   // UNICODE_TO_GBK[34826] := 16#8F38;
   // UNICODE_TO_GBK[34827] := 16#DD94;
   // UNICODE_TO_GBK[34828] := 16#8F39;
   // UNICODE_TO_GBK[34829] := 16#DD95;
   // UNICODE_TO_GBK[34830] := 16#8F3A;
   // UNICODE_TO_GBK[34831] := 16#DD96;
   // UNICODE_TO_GBK[34832] := 16#8F3B;
   // UNICODE_TO_GBK[34833] := 16#DD97;
   // UNICODE_TO_GBK[34834] := 16#8F3C;
   // UNICODE_TO_GBK[34835] := 16#DD98;
   // UNICODE_TO_GBK[34836] := 16#8F3D;
   // UNICODE_TO_GBK[34837] := 16#DD99;
   // UNICODE_TO_GBK[34838] := 16#8F3E;
   // UNICODE_TO_GBK[34839] := 16#DD9A;
   // UNICODE_TO_GBK[34840] := 16#8F3F;
   // UNICODE_TO_GBK[34841] := 16#DD9B;
   // UNICODE_TO_GBK[34842] := 16#8F40;
   // UNICODE_TO_GBK[34843] := 16#DD9C;
   // UNICODE_TO_GBK[34844] := 16#8F41;
   // UNICODE_TO_GBK[34845] := 16#DD9D;
   // UNICODE_TO_GBK[34846] := 16#8F42;
   // UNICODE_TO_GBK[34847] := 16#DD9E;
   // UNICODE_TO_GBK[34848] := 16#8F43;
   // UNICODE_TO_GBK[34849] := 16#DD9F;
   // UNICODE_TO_GBK[34850] := 16#8F44;
   // UNICODE_TO_GBK[34851] := 16#DDA0;
   // UNICODE_TO_GBK[34852] := 16#8F45;
   // UNICODE_TO_GBK[34853] := 16#DE40;
   // UNICODE_TO_GBK[34854] := 16#8F46;
   // UNICODE_TO_GBK[34855] := 16#DE41;
   // UNICODE_TO_GBK[34856] := 16#8F47;
   // UNICODE_TO_GBK[34857] := 16#DE42;
   // UNICODE_TO_GBK[34858] := 16#8F48;
   // UNICODE_TO_GBK[34859] := 16#DE43;
   // UNICODE_TO_GBK[34860] := 16#8F49;
   // UNICODE_TO_GBK[34861] := 16#DE44;
   // UNICODE_TO_GBK[34862] := 16#8F4A;
   // UNICODE_TO_GBK[34863] := 16#DE45;
   // UNICODE_TO_GBK[34864] := 16#8F4B;
   // UNICODE_TO_GBK[34865] := 16#DE46;
   // UNICODE_TO_GBK[34866] := 16#8F4C;
   // UNICODE_TO_GBK[34867] := 16#DE47;
   // UNICODE_TO_GBK[34868] := 16#8F4D;
   // UNICODE_TO_GBK[34869] := 16#DE48;
   // UNICODE_TO_GBK[34870] := 16#8F4E;
   // UNICODE_TO_GBK[34871] := 16#DE49;
   // UNICODE_TO_GBK[34872] := 16#8F4F;
   // UNICODE_TO_GBK[34873] := 16#DE4A;
   // UNICODE_TO_GBK[34874] := 16#8F50;
   // UNICODE_TO_GBK[34875] := 16#DE4B;
   // UNICODE_TO_GBK[34876] := 16#8F51;
   // UNICODE_TO_GBK[34877] := 16#DE4C;
   // UNICODE_TO_GBK[34878] := 16#8F52;
   // UNICODE_TO_GBK[34879] := 16#DE4D;
   // UNICODE_TO_GBK[34880] := 16#8F53;
   // UNICODE_TO_GBK[34881] := 16#DE4E;
   // UNICODE_TO_GBK[34882] := 16#8F54;
   // UNICODE_TO_GBK[34883] := 16#DE4F;
   // UNICODE_TO_GBK[34884] := 16#8F55;
   // UNICODE_TO_GBK[34885] := 16#DE50;
   // UNICODE_TO_GBK[34886] := 16#8F56;
   // UNICODE_TO_GBK[34887] := 16#DE51;
   // UNICODE_TO_GBK[34888] := 16#8F57;
   // UNICODE_TO_GBK[34889] := 16#DE52;
   // UNICODE_TO_GBK[34890] := 16#8F58;
   // UNICODE_TO_GBK[34891] := 16#DE53;
   // UNICODE_TO_GBK[34892] := 16#8F59;
   // UNICODE_TO_GBK[34893] := 16#DE54;
   // UNICODE_TO_GBK[34894] := 16#8F5A;
   // UNICODE_TO_GBK[34895] := 16#DE55;
   // UNICODE_TO_GBK[34896] := 16#8F5B;
   // UNICODE_TO_GBK[34897] := 16#DE56;
   // UNICODE_TO_GBK[34898] := 16#8F5C;
   // UNICODE_TO_GBK[34899] := 16#DE57;
   // UNICODE_TO_GBK[34900] := 16#8F5D;
   // UNICODE_TO_GBK[34901] := 16#DE58;
   // UNICODE_TO_GBK[34902] := 16#8F5E;
   // UNICODE_TO_GBK[34903] := 16#DE59;
   // UNICODE_TO_GBK[34904] := 16#8F5F;
   // UNICODE_TO_GBK[34905] := 16#DE5A;
   // UNICODE_TO_GBK[34906] := 16#8F60;
   // UNICODE_TO_GBK[34907] := 16#DE5B;
   // UNICODE_TO_GBK[34908] := 16#8F61;
   // UNICODE_TO_GBK[34909] := 16#DE5C;
   // UNICODE_TO_GBK[34910] := 16#8F62;
   // UNICODE_TO_GBK[34911] := 16#DE5D;
   // UNICODE_TO_GBK[34912] := 16#8F63;
   // UNICODE_TO_GBK[34913] := 16#DE5E;
   // UNICODE_TO_GBK[34914] := 16#8F64;
   // UNICODE_TO_GBK[34915] := 16#DE5F;
   // UNICODE_TO_GBK[34916] := 16#8F65;
   // UNICODE_TO_GBK[34917] := 16#DE60;
   // UNICODE_TO_GBK[34918] := 16#8F66;
   // UNICODE_TO_GBK[34919] := 16#B3B5;
   // UNICODE_TO_GBK[34920] := 16#8F67;
   // UNICODE_TO_GBK[34921] := 16#D4FE;
   // UNICODE_TO_GBK[34922] := 16#8F68;
   // UNICODE_TO_GBK[34923] := 16#B9EC;
   // UNICODE_TO_GBK[34924] := 16#8F69;
   // UNICODE_TO_GBK[34925] := 16#D0F9;
   // UNICODE_TO_GBK[34926] := 16#8F6A;
   // UNICODE_TO_GBK[34927] := 16#DE61;
   // UNICODE_TO_GBK[34928] := 16#8F6B;
   // UNICODE_TO_GBK[34929] := 16#E9ED;
   // UNICODE_TO_GBK[34930] := 16#8F6C;
   // UNICODE_TO_GBK[34931] := 16#D7AA;
   // UNICODE_TO_GBK[34932] := 16#8F6D;
   // UNICODE_TO_GBK[34933] := 16#E9EE;
   // UNICODE_TO_GBK[34934] := 16#8F6E;
   // UNICODE_TO_GBK[34935] := 16#C2D6;
   // UNICODE_TO_GBK[34936] := 16#8F6F;
   // UNICODE_TO_GBK[34937] := 16#C8ED;
   // UNICODE_TO_GBK[34938] := 16#8F70;
   // UNICODE_TO_GBK[34939] := 16#BAE4;
   // UNICODE_TO_GBK[34940] := 16#8F71;
   // UNICODE_TO_GBK[34941] := 16#E9EF;
   // UNICODE_TO_GBK[34942] := 16#8F72;
   // UNICODE_TO_GBK[34943] := 16#E9F0;
   // UNICODE_TO_GBK[34944] := 16#8F73;
   // UNICODE_TO_GBK[34945] := 16#E9F1;
   // UNICODE_TO_GBK[34946] := 16#8F74;
   // UNICODE_TO_GBK[34947] := 16#D6E1;
   // UNICODE_TO_GBK[34948] := 16#8F75;
   // UNICODE_TO_GBK[34949] := 16#E9F2;
   // UNICODE_TO_GBK[34950] := 16#8F76;
   // UNICODE_TO_GBK[34951] := 16#E9F3;
   // UNICODE_TO_GBK[34952] := 16#8F77;
   // UNICODE_TO_GBK[34953] := 16#E9F5;
   // UNICODE_TO_GBK[34954] := 16#8F78;
   // UNICODE_TO_GBK[34955] := 16#E9F4;
   // UNICODE_TO_GBK[34956] := 16#8F79;
   // UNICODE_TO_GBK[34957] := 16#E9F6;
   // UNICODE_TO_GBK[34958] := 16#8F7A;
   // UNICODE_TO_GBK[34959] := 16#E9F7;
   // UNICODE_TO_GBK[34960] := 16#8F7B;
   // UNICODE_TO_GBK[34961] := 16#C7E1;
   // UNICODE_TO_GBK[34962] := 16#8F7C;
   // UNICODE_TO_GBK[34963] := 16#E9F8;
   // UNICODE_TO_GBK[34964] := 16#8F7D;
   // UNICODE_TO_GBK[34965] := 16#D4D8;
   // UNICODE_TO_GBK[34966] := 16#8F7E;
   // UNICODE_TO_GBK[34967] := 16#E9F9;
   // UNICODE_TO_GBK[34968] := 16#8F7F;
   // UNICODE_TO_GBK[34969] := 16#BDCE;
   // UNICODE_TO_GBK[34970] := 16#8F80;
   // UNICODE_TO_GBK[34971] := 16#DE62;
   // UNICODE_TO_GBK[34972] := 16#8F81;
   // UNICODE_TO_GBK[34973] := 16#E9FA;
   // UNICODE_TO_GBK[34974] := 16#8F82;
   // UNICODE_TO_GBK[34975] := 16#E9FB;
   // UNICODE_TO_GBK[34976] := 16#8F83;
   // UNICODE_TO_GBK[34977] := 16#BDCF;
   // UNICODE_TO_GBK[34978] := 16#8F84;
   // UNICODE_TO_GBK[34979] := 16#E9FC;
   // UNICODE_TO_GBK[34980] := 16#8F85;
   // UNICODE_TO_GBK[34981] := 16#B8A8;
   // UNICODE_TO_GBK[34982] := 16#8F86;
   // UNICODE_TO_GBK[34983] := 16#C1BE;
   // UNICODE_TO_GBK[34984] := 16#8F87;
   // UNICODE_TO_GBK[34985] := 16#E9FD;
   // UNICODE_TO_GBK[34986] := 16#8F88;
   // UNICODE_TO_GBK[34987] := 16#B1B2;
   // UNICODE_TO_GBK[34988] := 16#8F89;
   // UNICODE_TO_GBK[34989] := 16#BBD4;
   // UNICODE_TO_GBK[34990] := 16#8F8A;
   // UNICODE_TO_GBK[34991] := 16#B9F5;
   // UNICODE_TO_GBK[34992] := 16#8F8B;
   // UNICODE_TO_GBK[34993] := 16#E9FE;
   // UNICODE_TO_GBK[34994] := 16#8F8C;
   // UNICODE_TO_GBK[34995] := 16#DE63;
   // UNICODE_TO_GBK[34996] := 16#8F8D;
   // UNICODE_TO_GBK[34997] := 16#EAA1;
   // UNICODE_TO_GBK[34998] := 16#8F8E;
   // UNICODE_TO_GBK[34999] := 16#EAA2;
   // UNICODE_TO_GBK[35000] := 16#8F8F;
   // UNICODE_TO_GBK[35001] := 16#EAA3;
   // UNICODE_TO_GBK[35002] := 16#8F90;
   // UNICODE_TO_GBK[35003] := 16#B7F8;
   // UNICODE_TO_GBK[35004] := 16#8F91;
   // UNICODE_TO_GBK[35005] := 16#BCAD;
   // UNICODE_TO_GBK[35006] := 16#8F92;
   // UNICODE_TO_GBK[35007] := 16#DE64;
   // UNICODE_TO_GBK[35008] := 16#8F93;
   // UNICODE_TO_GBK[35009] := 16#CAE4;
   // UNICODE_TO_GBK[35010] := 16#8F94;
   // UNICODE_TO_GBK[35011] := 16#E0CE;
   // UNICODE_TO_GBK[35012] := 16#8F95;
   // UNICODE_TO_GBK[35013] := 16#D4AF;
   // UNICODE_TO_GBK[35014] := 16#8F96;
   // UNICODE_TO_GBK[35015] := 16#CFBD;
   // UNICODE_TO_GBK[35016] := 16#8F97;
   // UNICODE_TO_GBK[35017] := 16#D5B7;
   // UNICODE_TO_GBK[35018] := 16#8F98;
   // UNICODE_TO_GBK[35019] := 16#EAA4;
   // UNICODE_TO_GBK[35020] := 16#8F99;
   // UNICODE_TO_GBK[35021] := 16#D5DE;
   // UNICODE_TO_GBK[35022] := 16#8F9A;
   // UNICODE_TO_GBK[35023] := 16#EAA5;
   // UNICODE_TO_GBK[35024] := 16#8F9B;
   // UNICODE_TO_GBK[35025] := 16#D0C1;
   // UNICODE_TO_GBK[35026] := 16#8F9C;
   // UNICODE_TO_GBK[35027] := 16#B9BC;
   // UNICODE_TO_GBK[35028] := 16#8F9D;
   // UNICODE_TO_GBK[35029] := 16#DE65;
   // UNICODE_TO_GBK[35030] := 16#8F9E;
   // UNICODE_TO_GBK[35031] := 16#B4C7;
   // UNICODE_TO_GBK[35032] := 16#8F9F;
   // UNICODE_TO_GBK[35033] := 16#B1D9;
   // UNICODE_TO_GBK[35034] := 16#8FA0;
   // UNICODE_TO_GBK[35035] := 16#DE66;
   // UNICODE_TO_GBK[35036] := 16#8FA1;
   // UNICODE_TO_GBK[35037] := 16#DE67;
   // UNICODE_TO_GBK[35038] := 16#8FA2;
   // UNICODE_TO_GBK[35039] := 16#DE68;
   // UNICODE_TO_GBK[35040] := 16#8FA3;
   // UNICODE_TO_GBK[35041] := 16#C0B1;
   // UNICODE_TO_GBK[35042] := 16#8FA4;
   // UNICODE_TO_GBK[35043] := 16#DE69;
   // UNICODE_TO_GBK[35044] := 16#8FA5;
   // UNICODE_TO_GBK[35045] := 16#DE6A;
   // UNICODE_TO_GBK[35046] := 16#8FA6;
   // UNICODE_TO_GBK[35047] := 16#DE6B;
   // UNICODE_TO_GBK[35048] := 16#8FA7;
   // UNICODE_TO_GBK[35049] := 16#DE6C;
   // UNICODE_TO_GBK[35050] := 16#8FA8;
   // UNICODE_TO_GBK[35051] := 16#B1E6;
   // UNICODE_TO_GBK[35052] := 16#8FA9;
   // UNICODE_TO_GBK[35053] := 16#B1E7;
   // UNICODE_TO_GBK[35054] := 16#8FAA;
   // UNICODE_TO_GBK[35055] := 16#DE6D;
   // UNICODE_TO_GBK[35056] := 16#8FAB;
   // UNICODE_TO_GBK[35057] := 16#B1E8;
   // UNICODE_TO_GBK[35058] := 16#8FAC;
   // UNICODE_TO_GBK[35059] := 16#DE6E;
   // UNICODE_TO_GBK[35060] := 16#8FAD;
   // UNICODE_TO_GBK[35061] := 16#DE6F;
   // UNICODE_TO_GBK[35062] := 16#8FAE;
   // UNICODE_TO_GBK[35063] := 16#DE70;
   // UNICODE_TO_GBK[35064] := 16#8FAF;
   // UNICODE_TO_GBK[35065] := 16#DE71;
   // UNICODE_TO_GBK[35066] := 16#8FB0;
   // UNICODE_TO_GBK[35067] := 16#B3BD;
   // UNICODE_TO_GBK[35068] := 16#8FB1;
   // UNICODE_TO_GBK[35069] := 16#C8E8;
   // UNICODE_TO_GBK[35070] := 16#8FB2;
   // UNICODE_TO_GBK[35071] := 16#DE72;
   // UNICODE_TO_GBK[35072] := 16#8FB3;
   // UNICODE_TO_GBK[35073] := 16#DE73;
   // UNICODE_TO_GBK[35074] := 16#8FB4;
   // UNICODE_TO_GBK[35075] := 16#DE74;
   // UNICODE_TO_GBK[35076] := 16#8FB5;
   // UNICODE_TO_GBK[35077] := 16#DE75;
   // UNICODE_TO_GBK[35078] := 16#8FB6;
   // UNICODE_TO_GBK[35079] := 16#E5C1;
   // UNICODE_TO_GBK[35080] := 16#8FB7;
   // UNICODE_TO_GBK[35081] := 16#DE76;
   // UNICODE_TO_GBK[35082] := 16#8FB8;
   // UNICODE_TO_GBK[35083] := 16#DE77;
   // UNICODE_TO_GBK[35084] := 16#8FB9;
   // UNICODE_TO_GBK[35085] := 16#B1DF;
   // UNICODE_TO_GBK[35086] := 16#8FBA;
   // UNICODE_TO_GBK[35087] := 16#DE78;
   // UNICODE_TO_GBK[35088] := 16#8FBB;
   // UNICODE_TO_GBK[35089] := 16#DE79;
   // UNICODE_TO_GBK[35090] := 16#8FBC;
   // UNICODE_TO_GBK[35091] := 16#DE7A;
   // UNICODE_TO_GBK[35092] := 16#8FBD;
   // UNICODE_TO_GBK[35093] := 16#C1C9;
   // UNICODE_TO_GBK[35094] := 16#8FBE;
   // UNICODE_TO_GBK[35095] := 16#B4EF;
   // UNICODE_TO_GBK[35096] := 16#8FBF;
   // UNICODE_TO_GBK[35097] := 16#DE7B;
   // UNICODE_TO_GBK[35098] := 16#8FC0;
   // UNICODE_TO_GBK[35099] := 16#DE7C;
   // UNICODE_TO_GBK[35100] := 16#8FC1;
   // UNICODE_TO_GBK[35101] := 16#C7A8;
   // UNICODE_TO_GBK[35102] := 16#8FC2;
   // UNICODE_TO_GBK[35103] := 16#D3D8;
   // UNICODE_TO_GBK[35104] := 16#8FC3;
   // UNICODE_TO_GBK[35105] := 16#DE7D;
   // UNICODE_TO_GBK[35106] := 16#8FC4;
   // UNICODE_TO_GBK[35107] := 16#C6F9;
   // UNICODE_TO_GBK[35108] := 16#8FC5;
   // UNICODE_TO_GBK[35109] := 16#D1B8;
   // UNICODE_TO_GBK[35110] := 16#8FC6;
   // UNICODE_TO_GBK[35111] := 16#DE7E;
   // UNICODE_TO_GBK[35112] := 16#8FC7;
   // UNICODE_TO_GBK[35113] := 16#B9FD;
   // UNICODE_TO_GBK[35114] := 16#8FC8;
   // UNICODE_TO_GBK[35115] := 16#C2F5;
   // UNICODE_TO_GBK[35116] := 16#8FC9;
   // UNICODE_TO_GBK[35117] := 16#DE80;
   // UNICODE_TO_GBK[35118] := 16#8FCA;
   // UNICODE_TO_GBK[35119] := 16#DE81;
   // UNICODE_TO_GBK[35120] := 16#8FCB;
   // UNICODE_TO_GBK[35121] := 16#DE82;
   // UNICODE_TO_GBK[35122] := 16#8FCC;
   // UNICODE_TO_GBK[35123] := 16#DE83;
   // UNICODE_TO_GBK[35124] := 16#8FCD;
   // UNICODE_TO_GBK[35125] := 16#DE84;
   // UNICODE_TO_GBK[35126] := 16#8FCE;
   // UNICODE_TO_GBK[35127] := 16#D3AD;
   // UNICODE_TO_GBK[35128] := 16#8FCF;
   // UNICODE_TO_GBK[35129] := 16#DE85;
   // UNICODE_TO_GBK[35130] := 16#8FD0;
   // UNICODE_TO_GBK[35131] := 16#D4CB;
   // UNICODE_TO_GBK[35132] := 16#8FD1;
   // UNICODE_TO_GBK[35133] := 16#BDFC;
   // UNICODE_TO_GBK[35134] := 16#8FD2;
   // UNICODE_TO_GBK[35135] := 16#DE86;
   // UNICODE_TO_GBK[35136] := 16#8FD3;
   // UNICODE_TO_GBK[35137] := 16#E5C2;
   // UNICODE_TO_GBK[35138] := 16#8FD4;
   // UNICODE_TO_GBK[35139] := 16#B7B5;
   // UNICODE_TO_GBK[35140] := 16#8FD5;
   // UNICODE_TO_GBK[35141] := 16#E5C3;
   // UNICODE_TO_GBK[35142] := 16#8FD6;
   // UNICODE_TO_GBK[35143] := 16#DE87;
   // UNICODE_TO_GBK[35144] := 16#8FD7;
   // UNICODE_TO_GBK[35145] := 16#DE88;
   // UNICODE_TO_GBK[35146] := 16#8FD8;
   // UNICODE_TO_GBK[35147] := 16#BBB9;
   // UNICODE_TO_GBK[35148] := 16#8FD9;
   // UNICODE_TO_GBK[35149] := 16#D5E2;
   // UNICODE_TO_GBK[35150] := 16#8FDA;
   // UNICODE_TO_GBK[35151] := 16#DE89;
   // UNICODE_TO_GBK[35152] := 16#8FDB;
   // UNICODE_TO_GBK[35153] := 16#BDF8;
   // UNICODE_TO_GBK[35154] := 16#8FDC;
   // UNICODE_TO_GBK[35155] := 16#D4B6;
   // UNICODE_TO_GBK[35156] := 16#8FDD;
   // UNICODE_TO_GBK[35157] := 16#CEA5;
   // UNICODE_TO_GBK[35158] := 16#8FDE;
   // UNICODE_TO_GBK[35159] := 16#C1AC;
   // UNICODE_TO_GBK[35160] := 16#8FDF;
   // UNICODE_TO_GBK[35161] := 16#B3D9;
   // UNICODE_TO_GBK[35162] := 16#8FE0;
   // UNICODE_TO_GBK[35163] := 16#DE8A;
   // UNICODE_TO_GBK[35164] := 16#8FE1;
   // UNICODE_TO_GBK[35165] := 16#DE8B;
   // UNICODE_TO_GBK[35166] := 16#8FE2;
   // UNICODE_TO_GBK[35167] := 16#CCF6;
   // UNICODE_TO_GBK[35168] := 16#8FE3;
   // UNICODE_TO_GBK[35169] := 16#DE8C;
   // UNICODE_TO_GBK[35170] := 16#8FE4;
   // UNICODE_TO_GBK[35171] := 16#E5C6;
   // UNICODE_TO_GBK[35172] := 16#8FE5;
   // UNICODE_TO_GBK[35173] := 16#E5C4;
   // UNICODE_TO_GBK[35174] := 16#8FE6;
   // UNICODE_TO_GBK[35175] := 16#E5C8;
   // UNICODE_TO_GBK[35176] := 16#8FE7;
   // UNICODE_TO_GBK[35177] := 16#DE8D;
   // UNICODE_TO_GBK[35178] := 16#8FE8;
   // UNICODE_TO_GBK[35179] := 16#E5CA;
   // UNICODE_TO_GBK[35180] := 16#8FE9;
   // UNICODE_TO_GBK[35181] := 16#E5C7;
   // UNICODE_TO_GBK[35182] := 16#8FEA;
   // UNICODE_TO_GBK[35183] := 16#B5CF;
   // UNICODE_TO_GBK[35184] := 16#8FEB;
   // UNICODE_TO_GBK[35185] := 16#C6C8;
   // UNICODE_TO_GBK[35186] := 16#8FEC;
   // UNICODE_TO_GBK[35187] := 16#DE8E;
   // UNICODE_TO_GBK[35188] := 16#8FED;
   // UNICODE_TO_GBK[35189] := 16#B5FC;
   // UNICODE_TO_GBK[35190] := 16#8FEE;
   // UNICODE_TO_GBK[35191] := 16#E5C5;
   // UNICODE_TO_GBK[35192] := 16#8FEF;
   // UNICODE_TO_GBK[35193] := 16#DE8F;
   // UNICODE_TO_GBK[35194] := 16#8FF0;
   // UNICODE_TO_GBK[35195] := 16#CAF6;
   // UNICODE_TO_GBK[35196] := 16#8FF1;
   // UNICODE_TO_GBK[35197] := 16#DE90;
   // UNICODE_TO_GBK[35198] := 16#8FF2;
   // UNICODE_TO_GBK[35199] := 16#DE91;
   // UNICODE_TO_GBK[35200] := 16#8FF3;
   // UNICODE_TO_GBK[35201] := 16#E5C9;
   // UNICODE_TO_GBK[35202] := 16#8FF4;
   // UNICODE_TO_GBK[35203] := 16#DE92;
   // UNICODE_TO_GBK[35204] := 16#8FF5;
   // UNICODE_TO_GBK[35205] := 16#DE93;
   // UNICODE_TO_GBK[35206] := 16#8FF6;
   // UNICODE_TO_GBK[35207] := 16#DE94;
   // UNICODE_TO_GBK[35208] := 16#8FF7;
   // UNICODE_TO_GBK[35209] := 16#C3D4;
   // UNICODE_TO_GBK[35210] := 16#8FF8;
   // UNICODE_TO_GBK[35211] := 16#B1C5;
   // UNICODE_TO_GBK[35212] := 16#8FF9;
   // UNICODE_TO_GBK[35213] := 16#BCA3;
   // UNICODE_TO_GBK[35214] := 16#8FFA;
   // UNICODE_TO_GBK[35215] := 16#DE95;
   // UNICODE_TO_GBK[35216] := 16#8FFB;
   // UNICODE_TO_GBK[35217] := 16#DE96;
   // UNICODE_TO_GBK[35218] := 16#8FFC;
   // UNICODE_TO_GBK[35219] := 16#DE97;
   // UNICODE_TO_GBK[35220] := 16#8FFD;
   // UNICODE_TO_GBK[35221] := 16#D7B7;
   // UNICODE_TO_GBK[35222] := 16#8FFE;
   // UNICODE_TO_GBK[35223] := 16#DE98;
   // UNICODE_TO_GBK[35224] := 16#8FFF;
   // UNICODE_TO_GBK[35225] := 16#DE99;
   // UNICODE_TO_GBK[35226] := 16#9000;
   // UNICODE_TO_GBK[35227] := 16#CDCB;
   // UNICODE_TO_GBK[35228] := 16#9001;
   // UNICODE_TO_GBK[35229] := 16#CBCD;
   // UNICODE_TO_GBK[35230] := 16#9002;
   // UNICODE_TO_GBK[35231] := 16#CACA;
   // UNICODE_TO_GBK[35232] := 16#9003;
   // UNICODE_TO_GBK[35233] := 16#CCD3;
   // UNICODE_TO_GBK[35234] := 16#9004;
   // UNICODE_TO_GBK[35235] := 16#E5CC;
   // UNICODE_TO_GBK[35236] := 16#9005;
   // UNICODE_TO_GBK[35237] := 16#E5CB;
   // UNICODE_TO_GBK[35238] := 16#9006;
   // UNICODE_TO_GBK[35239] := 16#C4E6;
   // UNICODE_TO_GBK[35240] := 16#9007;
   // UNICODE_TO_GBK[35241] := 16#DE9A;
   // UNICODE_TO_GBK[35242] := 16#9008;
   // UNICODE_TO_GBK[35243] := 16#DE9B;
   // UNICODE_TO_GBK[35244] := 16#9009;
   // UNICODE_TO_GBK[35245] := 16#D1A1;
   // UNICODE_TO_GBK[35246] := 16#900A;
   // UNICODE_TO_GBK[35247] := 16#D1B7;
   // UNICODE_TO_GBK[35248] := 16#900B;
   // UNICODE_TO_GBK[35249] := 16#E5CD;
   // UNICODE_TO_GBK[35250] := 16#900C;
   // UNICODE_TO_GBK[35251] := 16#DE9C;
   // UNICODE_TO_GBK[35252] := 16#900D;
   // UNICODE_TO_GBK[35253] := 16#E5D0;
   // UNICODE_TO_GBK[35254] := 16#900E;
   // UNICODE_TO_GBK[35255] := 16#DE9D;
   // UNICODE_TO_GBK[35256] := 16#900F;
   // UNICODE_TO_GBK[35257] := 16#CDB8;
   // UNICODE_TO_GBK[35258] := 16#9010;
   // UNICODE_TO_GBK[35259] := 16#D6F0;
   // UNICODE_TO_GBK[35260] := 16#9011;
   // UNICODE_TO_GBK[35261] := 16#E5CF;
   // UNICODE_TO_GBK[35262] := 16#9012;
   // UNICODE_TO_GBK[35263] := 16#B5DD;
   // UNICODE_TO_GBK[35264] := 16#9013;
   // UNICODE_TO_GBK[35265] := 16#DE9E;
   // UNICODE_TO_GBK[35266] := 16#9014;
   // UNICODE_TO_GBK[35267] := 16#CDBE;
   // UNICODE_TO_GBK[35268] := 16#9015;
   // UNICODE_TO_GBK[35269] := 16#DE9F;
   // UNICODE_TO_GBK[35270] := 16#9016;
   // UNICODE_TO_GBK[35271] := 16#E5D1;
   // UNICODE_TO_GBK[35272] := 16#9017;
   // UNICODE_TO_GBK[35273] := 16#B6BA;
   // UNICODE_TO_GBK[35274] := 16#9018;
   // UNICODE_TO_GBK[35275] := 16#DEA0;
   // UNICODE_TO_GBK[35276] := 16#9019;
   // UNICODE_TO_GBK[35277] := 16#DF40;
   // UNICODE_TO_GBK[35278] := 16#901A;
   // UNICODE_TO_GBK[35279] := 16#CDA8;
   // UNICODE_TO_GBK[35280] := 16#901B;
   // UNICODE_TO_GBK[35281] := 16#B9E4;
   // UNICODE_TO_GBK[35282] := 16#901C;
   // UNICODE_TO_GBK[35283] := 16#DF41;
   // UNICODE_TO_GBK[35284] := 16#901D;
   // UNICODE_TO_GBK[35285] := 16#CAC5;
   // UNICODE_TO_GBK[35286] := 16#901E;
   // UNICODE_TO_GBK[35287] := 16#B3D1;
   // UNICODE_TO_GBK[35288] := 16#901F;
   // UNICODE_TO_GBK[35289] := 16#CBD9;
   // UNICODE_TO_GBK[35290] := 16#9020;
   // UNICODE_TO_GBK[35291] := 16#D4EC;
   // UNICODE_TO_GBK[35292] := 16#9021;
   // UNICODE_TO_GBK[35293] := 16#E5D2;
   // UNICODE_TO_GBK[35294] := 16#9022;
   // UNICODE_TO_GBK[35295] := 16#B7EA;
   // UNICODE_TO_GBK[35296] := 16#9023;
   // UNICODE_TO_GBK[35297] := 16#DF42;
   // UNICODE_TO_GBK[35298] := 16#9024;
   // UNICODE_TO_GBK[35299] := 16#DF43;
   // UNICODE_TO_GBK[35300] := 16#9025;
   // UNICODE_TO_GBK[35301] := 16#DF44;
   // UNICODE_TO_GBK[35302] := 16#9026;
   // UNICODE_TO_GBK[35303] := 16#E5CE;
   // UNICODE_TO_GBK[35304] := 16#9027;
   // UNICODE_TO_GBK[35305] := 16#DF45;
   // UNICODE_TO_GBK[35306] := 16#9028;
   // UNICODE_TO_GBK[35307] := 16#DF46;
   // UNICODE_TO_GBK[35308] := 16#9029;
   // UNICODE_TO_GBK[35309] := 16#DF47;
   // UNICODE_TO_GBK[35310] := 16#902A;
   // UNICODE_TO_GBK[35311] := 16#DF48;
   // UNICODE_TO_GBK[35312] := 16#902B;
   // UNICODE_TO_GBK[35313] := 16#DF49;
   // UNICODE_TO_GBK[35314] := 16#902C;
   // UNICODE_TO_GBK[35315] := 16#DF4A;
   // UNICODE_TO_GBK[35316] := 16#902D;
   // UNICODE_TO_GBK[35317] := 16#E5D5;
   // UNICODE_TO_GBK[35318] := 16#902E;
   // UNICODE_TO_GBK[35319] := 16#B4FE;
   // UNICODE_TO_GBK[35320] := 16#902F;
   // UNICODE_TO_GBK[35321] := 16#E5D6;
   // UNICODE_TO_GBK[35322] := 16#9030;
   // UNICODE_TO_GBK[35323] := 16#DF4B;
   // UNICODE_TO_GBK[35324] := 16#9031;
   // UNICODE_TO_GBK[35325] := 16#DF4C;
   // UNICODE_TO_GBK[35326] := 16#9032;
   // UNICODE_TO_GBK[35327] := 16#DF4D;
   // UNICODE_TO_GBK[35328] := 16#9033;
   // UNICODE_TO_GBK[35329] := 16#DF4E;
   // UNICODE_TO_GBK[35330] := 16#9034;
   // UNICODE_TO_GBK[35331] := 16#DF4F;
   // UNICODE_TO_GBK[35332] := 16#9035;
   // UNICODE_TO_GBK[35333] := 16#E5D3;
   // UNICODE_TO_GBK[35334] := 16#9036;
   // UNICODE_TO_GBK[35335] := 16#E5D4;
   // UNICODE_TO_GBK[35336] := 16#9037;
   // UNICODE_TO_GBK[35337] := 16#DF50;
   // UNICODE_TO_GBK[35338] := 16#9038;
   // UNICODE_TO_GBK[35339] := 16#D2DD;
   // UNICODE_TO_GBK[35340] := 16#9039;
   // UNICODE_TO_GBK[35341] := 16#DF51;
   // UNICODE_TO_GBK[35342] := 16#903A;
   // UNICODE_TO_GBK[35343] := 16#DF52;
   // UNICODE_TO_GBK[35344] := 16#903B;
   // UNICODE_TO_GBK[35345] := 16#C2DF;
   // UNICODE_TO_GBK[35346] := 16#903C;
   // UNICODE_TO_GBK[35347] := 16#B1C6;
   // UNICODE_TO_GBK[35348] := 16#903D;
   // UNICODE_TO_GBK[35349] := 16#DF53;
   // UNICODE_TO_GBK[35350] := 16#903E;
   // UNICODE_TO_GBK[35351] := 16#D3E2;
   // UNICODE_TO_GBK[35352] := 16#903F;
   // UNICODE_TO_GBK[35353] := 16#DF54;
   // UNICODE_TO_GBK[35354] := 16#9040;
   // UNICODE_TO_GBK[35355] := 16#DF55;
   // UNICODE_TO_GBK[35356] := 16#9041;
   // UNICODE_TO_GBK[35357] := 16#B6DD;
   // UNICODE_TO_GBK[35358] := 16#9042;
   // UNICODE_TO_GBK[35359] := 16#CBEC;
   // UNICODE_TO_GBK[35360] := 16#9043;
   // UNICODE_TO_GBK[35361] := 16#DF56;
   // UNICODE_TO_GBK[35362] := 16#9044;
   // UNICODE_TO_GBK[35363] := 16#E5D7;
   // UNICODE_TO_GBK[35364] := 16#9045;
   // UNICODE_TO_GBK[35365] := 16#DF57;
   // UNICODE_TO_GBK[35366] := 16#9046;
   // UNICODE_TO_GBK[35367] := 16#DF58;
   // UNICODE_TO_GBK[35368] := 16#9047;
   // UNICODE_TO_GBK[35369] := 16#D3F6;
   // UNICODE_TO_GBK[35370] := 16#9048;
   // UNICODE_TO_GBK[35371] := 16#DF59;
   // UNICODE_TO_GBK[35372] := 16#9049;
   // UNICODE_TO_GBK[35373] := 16#DF5A;
   // UNICODE_TO_GBK[35374] := 16#904A;
   // UNICODE_TO_GBK[35375] := 16#DF5B;
   // UNICODE_TO_GBK[35376] := 16#904B;
   // UNICODE_TO_GBK[35377] := 16#DF5C;
   // UNICODE_TO_GBK[35378] := 16#904C;
   // UNICODE_TO_GBK[35379] := 16#DF5D;
   // UNICODE_TO_GBK[35380] := 16#904D;
   // UNICODE_TO_GBK[35381] := 16#B1E9;
   // UNICODE_TO_GBK[35382] := 16#904E;
   // UNICODE_TO_GBK[35383] := 16#DF5E;
   // UNICODE_TO_GBK[35384] := 16#904F;
   // UNICODE_TO_GBK[35385] := 16#B6F4;
   // UNICODE_TO_GBK[35386] := 16#9050;
   // UNICODE_TO_GBK[35387] := 16#E5DA;
   // UNICODE_TO_GBK[35388] := 16#9051;
   // UNICODE_TO_GBK[35389] := 16#E5D8;
   // UNICODE_TO_GBK[35390] := 16#9052;
   // UNICODE_TO_GBK[35391] := 16#E5D9;
   // UNICODE_TO_GBK[35392] := 16#9053;
   // UNICODE_TO_GBK[35393] := 16#B5C0;
   // UNICODE_TO_GBK[35394] := 16#9054;
   // UNICODE_TO_GBK[35395] := 16#DF5F;
   // UNICODE_TO_GBK[35396] := 16#9055;
   // UNICODE_TO_GBK[35397] := 16#DF60;
   // UNICODE_TO_GBK[35398] := 16#9056;
   // UNICODE_TO_GBK[35399] := 16#DF61;
   // UNICODE_TO_GBK[35400] := 16#9057;
   // UNICODE_TO_GBK[35401] := 16#D2C5;
   // UNICODE_TO_GBK[35402] := 16#9058;
   // UNICODE_TO_GBK[35403] := 16#E5DC;
   // UNICODE_TO_GBK[35404] := 16#9059;
   // UNICODE_TO_GBK[35405] := 16#DF62;
   // UNICODE_TO_GBK[35406] := 16#905A;
   // UNICODE_TO_GBK[35407] := 16#DF63;
   // UNICODE_TO_GBK[35408] := 16#905B;
   // UNICODE_TO_GBK[35409] := 16#E5DE;
   // UNICODE_TO_GBK[35410] := 16#905C;
   // UNICODE_TO_GBK[35411] := 16#DF64;
   // UNICODE_TO_GBK[35412] := 16#905D;
   // UNICODE_TO_GBK[35413] := 16#DF65;
   // UNICODE_TO_GBK[35414] := 16#905E;
   // UNICODE_TO_GBK[35415] := 16#DF66;
   // UNICODE_TO_GBK[35416] := 16#905F;
   // UNICODE_TO_GBK[35417] := 16#DF67;
   // UNICODE_TO_GBK[35418] := 16#9060;
   // UNICODE_TO_GBK[35419] := 16#DF68;
   // UNICODE_TO_GBK[35420] := 16#9061;
   // UNICODE_TO_GBK[35421] := 16#DF69;
   // UNICODE_TO_GBK[35422] := 16#9062;
   // UNICODE_TO_GBK[35423] := 16#E5DD;
   // UNICODE_TO_GBK[35424] := 16#9063;
   // UNICODE_TO_GBK[35425] := 16#C7B2;
   // UNICODE_TO_GBK[35426] := 16#9064;
   // UNICODE_TO_GBK[35427] := 16#DF6A;
   // UNICODE_TO_GBK[35428] := 16#9065;
   // UNICODE_TO_GBK[35429] := 16#D2A3;
   // UNICODE_TO_GBK[35430] := 16#9066;
   // UNICODE_TO_GBK[35431] := 16#DF6B;
   // UNICODE_TO_GBK[35432] := 16#9067;
   // UNICODE_TO_GBK[35433] := 16#DF6C;
   // UNICODE_TO_GBK[35434] := 16#9068;
   // UNICODE_TO_GBK[35435] := 16#E5DB;
   // UNICODE_TO_GBK[35436] := 16#9069;
   // UNICODE_TO_GBK[35437] := 16#DF6D;
   // UNICODE_TO_GBK[35438] := 16#906A;
   // UNICODE_TO_GBK[35439] := 16#DF6E;
   // UNICODE_TO_GBK[35440] := 16#906B;
   // UNICODE_TO_GBK[35441] := 16#DF6F;
   // UNICODE_TO_GBK[35442] := 16#906C;
   // UNICODE_TO_GBK[35443] := 16#DF70;
   // UNICODE_TO_GBK[35444] := 16#906D;
   // UNICODE_TO_GBK[35445] := 16#D4E2;
   // UNICODE_TO_GBK[35446] := 16#906E;
   // UNICODE_TO_GBK[35447] := 16#D5DA;
   // UNICODE_TO_GBK[35448] := 16#906F;
   // UNICODE_TO_GBK[35449] := 16#DF71;
   // UNICODE_TO_GBK[35450] := 16#9070;
   // UNICODE_TO_GBK[35451] := 16#DF72;
   // UNICODE_TO_GBK[35452] := 16#9071;
   // UNICODE_TO_GBK[35453] := 16#DF73;
   // UNICODE_TO_GBK[35454] := 16#9072;
   // UNICODE_TO_GBK[35455] := 16#DF74;
   // UNICODE_TO_GBK[35456] := 16#9073;
   // UNICODE_TO_GBK[35457] := 16#DF75;
   // UNICODE_TO_GBK[35458] := 16#9074;
   // UNICODE_TO_GBK[35459] := 16#E5E0;
   // UNICODE_TO_GBK[35460] := 16#9075;
   // UNICODE_TO_GBK[35461] := 16#D7F1;
   // UNICODE_TO_GBK[35462] := 16#9076;
   // UNICODE_TO_GBK[35463] := 16#DF76;
   // UNICODE_TO_GBK[35464] := 16#9077;
   // UNICODE_TO_GBK[35465] := 16#DF77;
   // UNICODE_TO_GBK[35466] := 16#9078;
   // UNICODE_TO_GBK[35467] := 16#DF78;
   // UNICODE_TO_GBK[35468] := 16#9079;
   // UNICODE_TO_GBK[35469] := 16#DF79;
   // UNICODE_TO_GBK[35470] := 16#907A;
   // UNICODE_TO_GBK[35471] := 16#DF7A;
   // UNICODE_TO_GBK[35472] := 16#907B;
   // UNICODE_TO_GBK[35473] := 16#DF7B;
   // UNICODE_TO_GBK[35474] := 16#907C;
   // UNICODE_TO_GBK[35475] := 16#DF7C;
   // UNICODE_TO_GBK[35476] := 16#907D;
   // UNICODE_TO_GBK[35477] := 16#E5E1;
   // UNICODE_TO_GBK[35478] := 16#907E;
   // UNICODE_TO_GBK[35479] := 16#DF7D;
   // UNICODE_TO_GBK[35480] := 16#907F;
   // UNICODE_TO_GBK[35481] := 16#B1DC;
   // UNICODE_TO_GBK[35482] := 16#9080;
   // UNICODE_TO_GBK[35483] := 16#D1FB;
   // UNICODE_TO_GBK[35484] := 16#9081;
   // UNICODE_TO_GBK[35485] := 16#DF7E;
   // UNICODE_TO_GBK[35486] := 16#9082;
   // UNICODE_TO_GBK[35487] := 16#E5E2;
   // UNICODE_TO_GBK[35488] := 16#9083;
   // UNICODE_TO_GBK[35489] := 16#E5E4;
   // UNICODE_TO_GBK[35490] := 16#9084;
   // UNICODE_TO_GBK[35491] := 16#DF80;
   // UNICODE_TO_GBK[35492] := 16#9085;
   // UNICODE_TO_GBK[35493] := 16#DF81;
   // UNICODE_TO_GBK[35494] := 16#9086;
   // UNICODE_TO_GBK[35495] := 16#DF82;
   // UNICODE_TO_GBK[35496] := 16#9087;
   // UNICODE_TO_GBK[35497] := 16#DF83;
   // UNICODE_TO_GBK[35498] := 16#9088;
   // UNICODE_TO_GBK[35499] := 16#E5E3;
   // UNICODE_TO_GBK[35500] := 16#9089;
   // UNICODE_TO_GBK[35501] := 16#DF84;
   // UNICODE_TO_GBK[35502] := 16#908A;
   // UNICODE_TO_GBK[35503] := 16#DF85;
   // UNICODE_TO_GBK[35504] := 16#908B;
   // UNICODE_TO_GBK[35505] := 16#E5E5;
   // UNICODE_TO_GBK[35506] := 16#908C;
   // UNICODE_TO_GBK[35507] := 16#DF86;
   // UNICODE_TO_GBK[35508] := 16#908D;
   // UNICODE_TO_GBK[35509] := 16#DF87;
   // UNICODE_TO_GBK[35510] := 16#908E;
   // UNICODE_TO_GBK[35511] := 16#DF88;
   // UNICODE_TO_GBK[35512] := 16#908F;
   // UNICODE_TO_GBK[35513] := 16#DF89;
   // UNICODE_TO_GBK[35514] := 16#9090;
   // UNICODE_TO_GBK[35515] := 16#DF8A;
   // UNICODE_TO_GBK[35516] := 16#9091;
   // UNICODE_TO_GBK[35517] := 16#D2D8;
   // UNICODE_TO_GBK[35518] := 16#9092;
   // UNICODE_TO_GBK[35519] := 16#DF8B;
   // UNICODE_TO_GBK[35520] := 16#9093;
   // UNICODE_TO_GBK[35521] := 16#B5CB;
   // UNICODE_TO_GBK[35522] := 16#9094;
   // UNICODE_TO_GBK[35523] := 16#DF8C;
   // UNICODE_TO_GBK[35524] := 16#9095;
   // UNICODE_TO_GBK[35525] := 16#E7DF;
   // UNICODE_TO_GBK[35526] := 16#9096;
   // UNICODE_TO_GBK[35527] := 16#DF8D;
   // UNICODE_TO_GBK[35528] := 16#9097;
   // UNICODE_TO_GBK[35529] := 16#DAF5;
   // UNICODE_TO_GBK[35530] := 16#9098;
   // UNICODE_TO_GBK[35531] := 16#DF8E;
   // UNICODE_TO_GBK[35532] := 16#9099;
   // UNICODE_TO_GBK[35533] := 16#DAF8;
   // UNICODE_TO_GBK[35534] := 16#909A;
   // UNICODE_TO_GBK[35535] := 16#DF8F;
   // UNICODE_TO_GBK[35536] := 16#909B;
   // UNICODE_TO_GBK[35537] := 16#DAF6;
   // UNICODE_TO_GBK[35538] := 16#909C;
   // UNICODE_TO_GBK[35539] := 16#DF90;
   // UNICODE_TO_GBK[35540] := 16#909D;
   // UNICODE_TO_GBK[35541] := 16#DAF7;
   // UNICODE_TO_GBK[35542] := 16#909E;
   // UNICODE_TO_GBK[35543] := 16#DF91;
   // UNICODE_TO_GBK[35544] := 16#909F;
   // UNICODE_TO_GBK[35545] := 16#DF92;
   // UNICODE_TO_GBK[35546] := 16#90A0;
   // UNICODE_TO_GBK[35547] := 16#DF93;
   // UNICODE_TO_GBK[35548] := 16#90A1;
   // UNICODE_TO_GBK[35549] := 16#DAFA;
   // UNICODE_TO_GBK[35550] := 16#90A2;
   // UNICODE_TO_GBK[35551] := 16#D0CF;
   // UNICODE_TO_GBK[35552] := 16#90A3;
   // UNICODE_TO_GBK[35553] := 16#C4C7;
   // UNICODE_TO_GBK[35554] := 16#90A4;
   // UNICODE_TO_GBK[35555] := 16#DF94;
   // UNICODE_TO_GBK[35556] := 16#90A5;
   // UNICODE_TO_GBK[35557] := 16#DF95;
   // UNICODE_TO_GBK[35558] := 16#90A6;
   // UNICODE_TO_GBK[35559] := 16#B0EE;
   // UNICODE_TO_GBK[35560] := 16#90A7;
   // UNICODE_TO_GBK[35561] := 16#DF96;
   // UNICODE_TO_GBK[35562] := 16#90A8;
   // UNICODE_TO_GBK[35563] := 16#DF97;
   // UNICODE_TO_GBK[35564] := 16#90A9;
   // UNICODE_TO_GBK[35565] := 16#DF98;
   // UNICODE_TO_GBK[35566] := 16#90AA;
   // UNICODE_TO_GBK[35567] := 16#D0B0;
   // UNICODE_TO_GBK[35568] := 16#90AB;
   // UNICODE_TO_GBK[35569] := 16#DF99;
   // UNICODE_TO_GBK[35570] := 16#90AC;
   // UNICODE_TO_GBK[35571] := 16#DAF9;
   // UNICODE_TO_GBK[35572] := 16#90AD;
   // UNICODE_TO_GBK[35573] := 16#DF9A;
   // UNICODE_TO_GBK[35574] := 16#90AE;
   // UNICODE_TO_GBK[35575] := 16#D3CA;
   // UNICODE_TO_GBK[35576] := 16#90AF;
   // UNICODE_TO_GBK[35577] := 16#BAAA;
   // UNICODE_TO_GBK[35578] := 16#90B0;
   // UNICODE_TO_GBK[35579] := 16#DBA2;
   // UNICODE_TO_GBK[35580] := 16#90B1;
   // UNICODE_TO_GBK[35581] := 16#C7F1;
   // UNICODE_TO_GBK[35582] := 16#90B2;
   // UNICODE_TO_GBK[35583] := 16#DF9B;
   // UNICODE_TO_GBK[35584] := 16#90B3;
   // UNICODE_TO_GBK[35585] := 16#DAFC;
   // UNICODE_TO_GBK[35586] := 16#90B4;
   // UNICODE_TO_GBK[35587] := 16#DAFB;
   // UNICODE_TO_GBK[35588] := 16#90B5;
   // UNICODE_TO_GBK[35589] := 16#C9DB;
   // UNICODE_TO_GBK[35590] := 16#90B6;
   // UNICODE_TO_GBK[35591] := 16#DAFD;
   // UNICODE_TO_GBK[35592] := 16#90B7;
   // UNICODE_TO_GBK[35593] := 16#DF9C;
   // UNICODE_TO_GBK[35594] := 16#90B8;
   // UNICODE_TO_GBK[35595] := 16#DBA1;
   // UNICODE_TO_GBK[35596] := 16#90B9;
   // UNICODE_TO_GBK[35597] := 16#D7DE;
   // UNICODE_TO_GBK[35598] := 16#90BA;
   // UNICODE_TO_GBK[35599] := 16#DAFE;
   // UNICODE_TO_GBK[35600] := 16#90BB;
   // UNICODE_TO_GBK[35601] := 16#C1DA;
   // UNICODE_TO_GBK[35602] := 16#90BC;
   // UNICODE_TO_GBK[35603] := 16#DF9D;
   // UNICODE_TO_GBK[35604] := 16#90BD;
   // UNICODE_TO_GBK[35605] := 16#DF9E;
   // UNICODE_TO_GBK[35606] := 16#90BE;
   // UNICODE_TO_GBK[35607] := 16#DBA5;
   // UNICODE_TO_GBK[35608] := 16#90BF;
   // UNICODE_TO_GBK[35609] := 16#DF9F;
   // UNICODE_TO_GBK[35610] := 16#90C0;
   // UNICODE_TO_GBK[35611] := 16#DFA0;
   // UNICODE_TO_GBK[35612] := 16#90C1;
   // UNICODE_TO_GBK[35613] := 16#D3F4;
   // UNICODE_TO_GBK[35614] := 16#90C2;
   // UNICODE_TO_GBK[35615] := 16#E040;
   // UNICODE_TO_GBK[35616] := 16#90C3;
   // UNICODE_TO_GBK[35617] := 16#E041;
   // UNICODE_TO_GBK[35618] := 16#90C4;
   // UNICODE_TO_GBK[35619] := 16#DBA7;
   // UNICODE_TO_GBK[35620] := 16#90C5;
   // UNICODE_TO_GBK[35621] := 16#DBA4;
   // UNICODE_TO_GBK[35622] := 16#90C6;
   // UNICODE_TO_GBK[35623] := 16#E042;
   // UNICODE_TO_GBK[35624] := 16#90C7;
   // UNICODE_TO_GBK[35625] := 16#DBA8;
   // UNICODE_TO_GBK[35626] := 16#90C8;
   // UNICODE_TO_GBK[35627] := 16#E043;
   // UNICODE_TO_GBK[35628] := 16#90C9;
   // UNICODE_TO_GBK[35629] := 16#E044;
   // UNICODE_TO_GBK[35630] := 16#90CA;
   // UNICODE_TO_GBK[35631] := 16#BDBC;
   // UNICODE_TO_GBK[35632] := 16#90CB;
   // UNICODE_TO_GBK[35633] := 16#E045;
   // UNICODE_TO_GBK[35634] := 16#90CC;
   // UNICODE_TO_GBK[35635] := 16#E046;
   // UNICODE_TO_GBK[35636] := 16#90CD;
   // UNICODE_TO_GBK[35637] := 16#E047;
   // UNICODE_TO_GBK[35638] := 16#90CE;
   // UNICODE_TO_GBK[35639] := 16#C0C9;
   // UNICODE_TO_GBK[35640] := 16#90CF;
   // UNICODE_TO_GBK[35641] := 16#DBA3;
   // UNICODE_TO_GBK[35642] := 16#90D0;
   // UNICODE_TO_GBK[35643] := 16#DBA6;
   // UNICODE_TO_GBK[35644] := 16#90D1;
   // UNICODE_TO_GBK[35645] := 16#D6A3;
   // UNICODE_TO_GBK[35646] := 16#90D2;
   // UNICODE_TO_GBK[35647] := 16#E048;
   // UNICODE_TO_GBK[35648] := 16#90D3;
   // UNICODE_TO_GBK[35649] := 16#DBA9;
   // UNICODE_TO_GBK[35650] := 16#90D4;
   // UNICODE_TO_GBK[35651] := 16#E049;
   // UNICODE_TO_GBK[35652] := 16#90D5;
   // UNICODE_TO_GBK[35653] := 16#E04A;
   // UNICODE_TO_GBK[35654] := 16#90D6;
   // UNICODE_TO_GBK[35655] := 16#E04B;
   // UNICODE_TO_GBK[35656] := 16#90D7;
   // UNICODE_TO_GBK[35657] := 16#DBAD;
   // UNICODE_TO_GBK[35658] := 16#90D8;
   // UNICODE_TO_GBK[35659] := 16#E04C;
   // UNICODE_TO_GBK[35660] := 16#90D9;
   // UNICODE_TO_GBK[35661] := 16#E04D;
   // UNICODE_TO_GBK[35662] := 16#90DA;
   // UNICODE_TO_GBK[35663] := 16#E04E;
   // UNICODE_TO_GBK[35664] := 16#90DB;
   // UNICODE_TO_GBK[35665] := 16#DBAE;
   // UNICODE_TO_GBK[35666] := 16#90DC;
   // UNICODE_TO_GBK[35667] := 16#DBAC;
   // UNICODE_TO_GBK[35668] := 16#90DD;
   // UNICODE_TO_GBK[35669] := 16#BAC2;
   // UNICODE_TO_GBK[35670] := 16#90DE;
   // UNICODE_TO_GBK[35671] := 16#E04F;
   // UNICODE_TO_GBK[35672] := 16#90DF;
   // UNICODE_TO_GBK[35673] := 16#E050;
   // UNICODE_TO_GBK[35674] := 16#90E0;
   // UNICODE_TO_GBK[35675] := 16#E051;
   // UNICODE_TO_GBK[35676] := 16#90E1;
   // UNICODE_TO_GBK[35677] := 16#BFA4;
   // UNICODE_TO_GBK[35678] := 16#90E2;
   // UNICODE_TO_GBK[35679] := 16#DBAB;
   // UNICODE_TO_GBK[35680] := 16#90E3;
   // UNICODE_TO_GBK[35681] := 16#E052;
   // UNICODE_TO_GBK[35682] := 16#90E4;
   // UNICODE_TO_GBK[35683] := 16#E053;
   // UNICODE_TO_GBK[35684] := 16#90E5;
   // UNICODE_TO_GBK[35685] := 16#E054;
   // UNICODE_TO_GBK[35686] := 16#90E6;
   // UNICODE_TO_GBK[35687] := 16#DBAA;
   // UNICODE_TO_GBK[35688] := 16#90E7;
   // UNICODE_TO_GBK[35689] := 16#D4C7;
   // UNICODE_TO_GBK[35690] := 16#90E8;
   // UNICODE_TO_GBK[35691] := 16#B2BF;
   // UNICODE_TO_GBK[35692] := 16#90E9;
   // UNICODE_TO_GBK[35693] := 16#E055;
   // UNICODE_TO_GBK[35694] := 16#90EA;
   // UNICODE_TO_GBK[35695] := 16#E056;
   // UNICODE_TO_GBK[35696] := 16#90EB;
   // UNICODE_TO_GBK[35697] := 16#DBAF;
   // UNICODE_TO_GBK[35698] := 16#90EC;
   // UNICODE_TO_GBK[35699] := 16#E057;
   // UNICODE_TO_GBK[35700] := 16#90ED;
   // UNICODE_TO_GBK[35701] := 16#B9F9;
   // UNICODE_TO_GBK[35702] := 16#90EE;
   // UNICODE_TO_GBK[35703] := 16#E058;
   // UNICODE_TO_GBK[35704] := 16#90EF;
   // UNICODE_TO_GBK[35705] := 16#DBB0;
   // UNICODE_TO_GBK[35706] := 16#90F0;
   // UNICODE_TO_GBK[35707] := 16#E059;
   // UNICODE_TO_GBK[35708] := 16#90F1;
   // UNICODE_TO_GBK[35709] := 16#E05A;
   // UNICODE_TO_GBK[35710] := 16#90F2;
   // UNICODE_TO_GBK[35711] := 16#E05B;
   // UNICODE_TO_GBK[35712] := 16#90F3;
   // UNICODE_TO_GBK[35713] := 16#E05C;
   // UNICODE_TO_GBK[35714] := 16#90F4;
   // UNICODE_TO_GBK[35715] := 16#B3BB;
   // UNICODE_TO_GBK[35716] := 16#90F5;
   // UNICODE_TO_GBK[35717] := 16#E05D;
   // UNICODE_TO_GBK[35718] := 16#90F6;
   // UNICODE_TO_GBK[35719] := 16#E05E;
   // UNICODE_TO_GBK[35720] := 16#90F7;
   // UNICODE_TO_GBK[35721] := 16#E05F;
   // UNICODE_TO_GBK[35722] := 16#90F8;
   // UNICODE_TO_GBK[35723] := 16#B5A6;
   // UNICODE_TO_GBK[35724] := 16#90F9;
   // UNICODE_TO_GBK[35725] := 16#E060;
   // UNICODE_TO_GBK[35726] := 16#90FA;
   // UNICODE_TO_GBK[35727] := 16#E061;
   // UNICODE_TO_GBK[35728] := 16#90FB;
   // UNICODE_TO_GBK[35729] := 16#E062;
   // UNICODE_TO_GBK[35730] := 16#90FC;
   // UNICODE_TO_GBK[35731] := 16#E063;
   // UNICODE_TO_GBK[35732] := 16#90FD;
   // UNICODE_TO_GBK[35733] := 16#B6BC;
   // UNICODE_TO_GBK[35734] := 16#90FE;
   // UNICODE_TO_GBK[35735] := 16#DBB1;
   // UNICODE_TO_GBK[35736] := 16#90FF;
   // UNICODE_TO_GBK[35737] := 16#E064;
   // UNICODE_TO_GBK[35738] := 16#9100;
   // UNICODE_TO_GBK[35739] := 16#E065;
   // UNICODE_TO_GBK[35740] := 16#9101;
   // UNICODE_TO_GBK[35741] := 16#E066;
   // UNICODE_TO_GBK[35742] := 16#9102;
   // UNICODE_TO_GBK[35743] := 16#B6F5;
   // UNICODE_TO_GBK[35744] := 16#9103;
   // UNICODE_TO_GBK[35745] := 16#E067;
   // UNICODE_TO_GBK[35746] := 16#9104;
   // UNICODE_TO_GBK[35747] := 16#DBB2;
   // UNICODE_TO_GBK[35748] := 16#9105;
   // UNICODE_TO_GBK[35749] := 16#E068;
   // UNICODE_TO_GBK[35750] := 16#9106;
   // UNICODE_TO_GBK[35751] := 16#E069;
   // UNICODE_TO_GBK[35752] := 16#9107;
   // UNICODE_TO_GBK[35753] := 16#E06A;
   // UNICODE_TO_GBK[35754] := 16#9108;
   // UNICODE_TO_GBK[35755] := 16#E06B;
   // UNICODE_TO_GBK[35756] := 16#9109;
   // UNICODE_TO_GBK[35757] := 16#E06C;
   // UNICODE_TO_GBK[35758] := 16#910A;
   // UNICODE_TO_GBK[35759] := 16#E06D;
   // UNICODE_TO_GBK[35760] := 16#910B;
   // UNICODE_TO_GBK[35761] := 16#E06E;
   // UNICODE_TO_GBK[35762] := 16#910C;
   // UNICODE_TO_GBK[35763] := 16#E06F;
   // UNICODE_TO_GBK[35764] := 16#910D;
   // UNICODE_TO_GBK[35765] := 16#E070;
   // UNICODE_TO_GBK[35766] := 16#910E;
   // UNICODE_TO_GBK[35767] := 16#E071;
   // UNICODE_TO_GBK[35768] := 16#910F;
   // UNICODE_TO_GBK[35769] := 16#E072;
   // UNICODE_TO_GBK[35770] := 16#9110;
   // UNICODE_TO_GBK[35771] := 16#E073;
   // UNICODE_TO_GBK[35772] := 16#9111;
   // UNICODE_TO_GBK[35773] := 16#E074;
   // UNICODE_TO_GBK[35774] := 16#9112;
   // UNICODE_TO_GBK[35775] := 16#E075;
   // UNICODE_TO_GBK[35776] := 16#9113;
   // UNICODE_TO_GBK[35777] := 16#E076;
   // UNICODE_TO_GBK[35778] := 16#9114;
   // UNICODE_TO_GBK[35779] := 16#E077;
   // UNICODE_TO_GBK[35780] := 16#9115;
   // UNICODE_TO_GBK[35781] := 16#E078;
   // UNICODE_TO_GBK[35782] := 16#9116;
   // UNICODE_TO_GBK[35783] := 16#E079;
   // UNICODE_TO_GBK[35784] := 16#9117;
   // UNICODE_TO_GBK[35785] := 16#E07A;
   // UNICODE_TO_GBK[35786] := 16#9118;
   // UNICODE_TO_GBK[35787] := 16#E07B;
   // UNICODE_TO_GBK[35788] := 16#9119;
   // UNICODE_TO_GBK[35789] := 16#B1C9;
   // UNICODE_TO_GBK[35790] := 16#911A;
   // UNICODE_TO_GBK[35791] := 16#E07C;
   // UNICODE_TO_GBK[35792] := 16#911B;
   // UNICODE_TO_GBK[35793] := 16#E07D;
   // UNICODE_TO_GBK[35794] := 16#911C;
   // UNICODE_TO_GBK[35795] := 16#E07E;
   // UNICODE_TO_GBK[35796] := 16#911D;
   // UNICODE_TO_GBK[35797] := 16#E080;
   // UNICODE_TO_GBK[35798] := 16#911E;
   // UNICODE_TO_GBK[35799] := 16#DBB4;
   // UNICODE_TO_GBK[35800] := 16#911F;
   // UNICODE_TO_GBK[35801] := 16#E081;
   // UNICODE_TO_GBK[35802] := 16#9120;
   // UNICODE_TO_GBK[35803] := 16#E082;
   // UNICODE_TO_GBK[35804] := 16#9121;
   // UNICODE_TO_GBK[35805] := 16#E083;
   // UNICODE_TO_GBK[35806] := 16#9122;
   // UNICODE_TO_GBK[35807] := 16#DBB3;
   // UNICODE_TO_GBK[35808] := 16#9123;
   // UNICODE_TO_GBK[35809] := 16#DBB5;
   // UNICODE_TO_GBK[35810] := 16#9124;
   // UNICODE_TO_GBK[35811] := 16#E084;
   // UNICODE_TO_GBK[35812] := 16#9125;
   // UNICODE_TO_GBK[35813] := 16#E085;
   // UNICODE_TO_GBK[35814] := 16#9126;
   // UNICODE_TO_GBK[35815] := 16#E086;
   // UNICODE_TO_GBK[35816] := 16#9127;
   // UNICODE_TO_GBK[35817] := 16#E087;
   // UNICODE_TO_GBK[35818] := 16#9128;
   // UNICODE_TO_GBK[35819] := 16#E088;
   // UNICODE_TO_GBK[35820] := 16#9129;
   // UNICODE_TO_GBK[35821] := 16#E089;
   // UNICODE_TO_GBK[35822] := 16#912A;
   // UNICODE_TO_GBK[35823] := 16#E08A;
   // UNICODE_TO_GBK[35824] := 16#912B;
   // UNICODE_TO_GBK[35825] := 16#E08B;
   // UNICODE_TO_GBK[35826] := 16#912C;
   // UNICODE_TO_GBK[35827] := 16#E08C;
   // UNICODE_TO_GBK[35828] := 16#912D;
   // UNICODE_TO_GBK[35829] := 16#E08D;
   // UNICODE_TO_GBK[35830] := 16#912E;
   // UNICODE_TO_GBK[35831] := 16#E08E;
   // UNICODE_TO_GBK[35832] := 16#912F;
   // UNICODE_TO_GBK[35833] := 16#DBB7;
   // UNICODE_TO_GBK[35834] := 16#9130;
   // UNICODE_TO_GBK[35835] := 16#E08F;
   // UNICODE_TO_GBK[35836] := 16#9131;
   // UNICODE_TO_GBK[35837] := 16#DBB6;
   // UNICODE_TO_GBK[35838] := 16#9132;
   // UNICODE_TO_GBK[35839] := 16#E090;
   // UNICODE_TO_GBK[35840] := 16#9133;
   // UNICODE_TO_GBK[35841] := 16#E091;
   // UNICODE_TO_GBK[35842] := 16#9134;
   // UNICODE_TO_GBK[35843] := 16#E092;
   // UNICODE_TO_GBK[35844] := 16#9135;
   // UNICODE_TO_GBK[35845] := 16#E093;
   // UNICODE_TO_GBK[35846] := 16#9136;
   // UNICODE_TO_GBK[35847] := 16#E094;
   // UNICODE_TO_GBK[35848] := 16#9137;
   // UNICODE_TO_GBK[35849] := 16#E095;
   // UNICODE_TO_GBK[35850] := 16#9138;
   // UNICODE_TO_GBK[35851] := 16#E096;
   // UNICODE_TO_GBK[35852] := 16#9139;
   // UNICODE_TO_GBK[35853] := 16#DBB8;
   // UNICODE_TO_GBK[35854] := 16#913A;
   // UNICODE_TO_GBK[35855] := 16#E097;
   // UNICODE_TO_GBK[35856] := 16#913B;
   // UNICODE_TO_GBK[35857] := 16#E098;
   // UNICODE_TO_GBK[35858] := 16#913C;
   // UNICODE_TO_GBK[35859] := 16#E099;
   // UNICODE_TO_GBK[35860] := 16#913D;
   // UNICODE_TO_GBK[35861] := 16#E09A;
   // UNICODE_TO_GBK[35862] := 16#913E;
   // UNICODE_TO_GBK[35863] := 16#E09B;
   // UNICODE_TO_GBK[35864] := 16#913F;
   // UNICODE_TO_GBK[35865] := 16#E09C;
   // UNICODE_TO_GBK[35866] := 16#9140;
   // UNICODE_TO_GBK[35867] := 16#E09D;
   // UNICODE_TO_GBK[35868] := 16#9141;
   // UNICODE_TO_GBK[35869] := 16#E09E;
   // UNICODE_TO_GBK[35870] := 16#9142;
   // UNICODE_TO_GBK[35871] := 16#E09F;
   // UNICODE_TO_GBK[35872] := 16#9143;
   // UNICODE_TO_GBK[35873] := 16#DBB9;
   // UNICODE_TO_GBK[35874] := 16#9144;
   // UNICODE_TO_GBK[35875] := 16#E0A0;
   // UNICODE_TO_GBK[35876] := 16#9145;
   // UNICODE_TO_GBK[35877] := 16#E140;
   // UNICODE_TO_GBK[35878] := 16#9146;
   // UNICODE_TO_GBK[35879] := 16#DBBA;
   // UNICODE_TO_GBK[35880] := 16#9147;
   // UNICODE_TO_GBK[35881] := 16#E141;
   // UNICODE_TO_GBK[35882] := 16#9148;
   // UNICODE_TO_GBK[35883] := 16#E142;
   // UNICODE_TO_GBK[35884] := 16#9149;
   // UNICODE_TO_GBK[35885] := 16#D3CF;
   // UNICODE_TO_GBK[35886] := 16#914A;
   // UNICODE_TO_GBK[35887] := 16#F4FA;
   // UNICODE_TO_GBK[35888] := 16#914B;
   // UNICODE_TO_GBK[35889] := 16#C7F5;
   // UNICODE_TO_GBK[35890] := 16#914C;
   // UNICODE_TO_GBK[35891] := 16#D7C3;
   // UNICODE_TO_GBK[35892] := 16#914D;
   // UNICODE_TO_GBK[35893] := 16#C5E4;
   // UNICODE_TO_GBK[35894] := 16#914E;
   // UNICODE_TO_GBK[35895] := 16#F4FC;
   // UNICODE_TO_GBK[35896] := 16#914F;
   // UNICODE_TO_GBK[35897] := 16#F4FD;
   // UNICODE_TO_GBK[35898] := 16#9150;
   // UNICODE_TO_GBK[35899] := 16#F4FB;
   // UNICODE_TO_GBK[35900] := 16#9151;
   // UNICODE_TO_GBK[35901] := 16#E143;
   // UNICODE_TO_GBK[35902] := 16#9152;
   // UNICODE_TO_GBK[35903] := 16#BEC6;
   // UNICODE_TO_GBK[35904] := 16#9153;
   // UNICODE_TO_GBK[35905] := 16#E144;
   // UNICODE_TO_GBK[35906] := 16#9154;
   // UNICODE_TO_GBK[35907] := 16#E145;
   // UNICODE_TO_GBK[35908] := 16#9155;
   // UNICODE_TO_GBK[35909] := 16#E146;
   // UNICODE_TO_GBK[35910] := 16#9156;
   // UNICODE_TO_GBK[35911] := 16#E147;
   // UNICODE_TO_GBK[35912] := 16#9157;
   // UNICODE_TO_GBK[35913] := 16#D0EF;
   // UNICODE_TO_GBK[35914] := 16#9158;
   // UNICODE_TO_GBK[35915] := 16#E148;
   // UNICODE_TO_GBK[35916] := 16#9159;
   // UNICODE_TO_GBK[35917] := 16#E149;
   // UNICODE_TO_GBK[35918] := 16#915A;
   // UNICODE_TO_GBK[35919] := 16#B7D3;
   // UNICODE_TO_GBK[35920] := 16#915B;
   // UNICODE_TO_GBK[35921] := 16#E14A;
   // UNICODE_TO_GBK[35922] := 16#915C;
   // UNICODE_TO_GBK[35923] := 16#E14B;
   // UNICODE_TO_GBK[35924] := 16#915D;
   // UNICODE_TO_GBK[35925] := 16#D4CD;
   // UNICODE_TO_GBK[35926] := 16#915E;
   // UNICODE_TO_GBK[35927] := 16#CCAA;
   // UNICODE_TO_GBK[35928] := 16#915F;
   // UNICODE_TO_GBK[35929] := 16#E14C;
   // UNICODE_TO_GBK[35930] := 16#9160;
   // UNICODE_TO_GBK[35931] := 16#E14D;
   // UNICODE_TO_GBK[35932] := 16#9161;
   // UNICODE_TO_GBK[35933] := 16#F5A2;
   // UNICODE_TO_GBK[35934] := 16#9162;
   // UNICODE_TO_GBK[35935] := 16#F5A1;
   // UNICODE_TO_GBK[35936] := 16#9163;
   // UNICODE_TO_GBK[35937] := 16#BAA8;
   // UNICODE_TO_GBK[35938] := 16#9164;
   // UNICODE_TO_GBK[35939] := 16#F4FE;
   // UNICODE_TO_GBK[35940] := 16#9165;
   // UNICODE_TO_GBK[35941] := 16#CBD6;
   // UNICODE_TO_GBK[35942] := 16#9166;
   // UNICODE_TO_GBK[35943] := 16#E14E;
   // UNICODE_TO_GBK[35944] := 16#9167;
   // UNICODE_TO_GBK[35945] := 16#E14F;
   // UNICODE_TO_GBK[35946] := 16#9168;
   // UNICODE_TO_GBK[35947] := 16#E150;
   // UNICODE_TO_GBK[35948] := 16#9169;
   // UNICODE_TO_GBK[35949] := 16#F5A4;
   // UNICODE_TO_GBK[35950] := 16#916A;
   // UNICODE_TO_GBK[35951] := 16#C0D2;
   // UNICODE_TO_GBK[35952] := 16#916B;
   // UNICODE_TO_GBK[35953] := 16#E151;
   // UNICODE_TO_GBK[35954] := 16#916C;
   // UNICODE_TO_GBK[35955] := 16#B3EA;
   // UNICODE_TO_GBK[35956] := 16#916D;
   // UNICODE_TO_GBK[35957] := 16#E152;
   // UNICODE_TO_GBK[35958] := 16#916E;
   // UNICODE_TO_GBK[35959] := 16#CDAA;
   // UNICODE_TO_GBK[35960] := 16#916F;
   // UNICODE_TO_GBK[35961] := 16#F5A5;
   // UNICODE_TO_GBK[35962] := 16#9170;
   // UNICODE_TO_GBK[35963] := 16#F5A3;
   // UNICODE_TO_GBK[35964] := 16#9171;
   // UNICODE_TO_GBK[35965] := 16#BDB4;
   // UNICODE_TO_GBK[35966] := 16#9172;
   // UNICODE_TO_GBK[35967] := 16#F5A8;
   // UNICODE_TO_GBK[35968] := 16#9173;
   // UNICODE_TO_GBK[35969] := 16#E153;
   // UNICODE_TO_GBK[35970] := 16#9174;
   // UNICODE_TO_GBK[35971] := 16#F5A9;
   // UNICODE_TO_GBK[35972] := 16#9175;
   // UNICODE_TO_GBK[35973] := 16#BDCD;
   // UNICODE_TO_GBK[35974] := 16#9176;
   // UNICODE_TO_GBK[35975] := 16#C3B8;
   // UNICODE_TO_GBK[35976] := 16#9177;
   // UNICODE_TO_GBK[35977] := 16#BFE1;
   // UNICODE_TO_GBK[35978] := 16#9178;
   // UNICODE_TO_GBK[35979] := 16#CBE1;
   // UNICODE_TO_GBK[35980] := 16#9179;
   // UNICODE_TO_GBK[35981] := 16#F5AA;
   // UNICODE_TO_GBK[35982] := 16#917A;
   // UNICODE_TO_GBK[35983] := 16#E154;
   // UNICODE_TO_GBK[35984] := 16#917B;
   // UNICODE_TO_GBK[35985] := 16#E155;
   // UNICODE_TO_GBK[35986] := 16#917C;
   // UNICODE_TO_GBK[35987] := 16#E156;
   // UNICODE_TO_GBK[35988] := 16#917D;
   // UNICODE_TO_GBK[35989] := 16#F5A6;
   // UNICODE_TO_GBK[35990] := 16#917E;
   // UNICODE_TO_GBK[35991] := 16#F5A7;
   // UNICODE_TO_GBK[35992] := 16#917F;
   // UNICODE_TO_GBK[35993] := 16#C4F0;
   // UNICODE_TO_GBK[35994] := 16#9180;
   // UNICODE_TO_GBK[35995] := 16#E157;
   // UNICODE_TO_GBK[35996] := 16#9181;
   // UNICODE_TO_GBK[35997] := 16#E158;
   // UNICODE_TO_GBK[35998] := 16#9182;
   // UNICODE_TO_GBK[35999] := 16#E159;
   // UNICODE_TO_GBK[36000] := 16#9183;
   // UNICODE_TO_GBK[36001] := 16#E15A;
   // UNICODE_TO_GBK[36002] := 16#9184;
   // UNICODE_TO_GBK[36003] := 16#E15B;
   // UNICODE_TO_GBK[36004] := 16#9185;
   // UNICODE_TO_GBK[36005] := 16#F5AC;
   // UNICODE_TO_GBK[36006] := 16#9186;
   // UNICODE_TO_GBK[36007] := 16#E15C;
   // UNICODE_TO_GBK[36008] := 16#9187;
   // UNICODE_TO_GBK[36009] := 16#B4BC;
   // UNICODE_TO_GBK[36010] := 16#9188;
   // UNICODE_TO_GBK[36011] := 16#E15D;
   // UNICODE_TO_GBK[36012] := 16#9189;
   // UNICODE_TO_GBK[36013] := 16#D7ED;
   // UNICODE_TO_GBK[36014] := 16#918A;
   // UNICODE_TO_GBK[36015] := 16#E15E;
   // UNICODE_TO_GBK[36016] := 16#918B;
   // UNICODE_TO_GBK[36017] := 16#B4D7;
   // UNICODE_TO_GBK[36018] := 16#918C;
   // UNICODE_TO_GBK[36019] := 16#F5AB;
   // UNICODE_TO_GBK[36020] := 16#918D;
   // UNICODE_TO_GBK[36021] := 16#F5AE;
   // UNICODE_TO_GBK[36022] := 16#918E;
   // UNICODE_TO_GBK[36023] := 16#E15F;
   // UNICODE_TO_GBK[36024] := 16#918F;
   // UNICODE_TO_GBK[36025] := 16#E160;
   // UNICODE_TO_GBK[36026] := 16#9190;
   // UNICODE_TO_GBK[36027] := 16#F5AD;
   // UNICODE_TO_GBK[36028] := 16#9191;
   // UNICODE_TO_GBK[36029] := 16#F5AF;
   // UNICODE_TO_GBK[36030] := 16#9192;
   // UNICODE_TO_GBK[36031] := 16#D0D1;
   // UNICODE_TO_GBK[36032] := 16#9193;
   // UNICODE_TO_GBK[36033] := 16#E161;
   // UNICODE_TO_GBK[36034] := 16#9194;
   // UNICODE_TO_GBK[36035] := 16#E162;
   // UNICODE_TO_GBK[36036] := 16#9195;
   // UNICODE_TO_GBK[36037] := 16#E163;
   // UNICODE_TO_GBK[36038] := 16#9196;
   // UNICODE_TO_GBK[36039] := 16#E164;
   // UNICODE_TO_GBK[36040] := 16#9197;
   // UNICODE_TO_GBK[36041] := 16#E165;
   // UNICODE_TO_GBK[36042] := 16#9198;
   // UNICODE_TO_GBK[36043] := 16#E166;
   // UNICODE_TO_GBK[36044] := 16#9199;
   // UNICODE_TO_GBK[36045] := 16#E167;
   // UNICODE_TO_GBK[36046] := 16#919A;
   // UNICODE_TO_GBK[36047] := 16#C3D1;
   // UNICODE_TO_GBK[36048] := 16#919B;
   // UNICODE_TO_GBK[36049] := 16#C8A9;
   // UNICODE_TO_GBK[36050] := 16#919C;
   // UNICODE_TO_GBK[36051] := 16#E168;
   // UNICODE_TO_GBK[36052] := 16#919D;
   // UNICODE_TO_GBK[36053] := 16#E169;
   // UNICODE_TO_GBK[36054] := 16#919E;
   // UNICODE_TO_GBK[36055] := 16#E16A;
   // UNICODE_TO_GBK[36056] := 16#919F;
   // UNICODE_TO_GBK[36057] := 16#E16B;
   // UNICODE_TO_GBK[36058] := 16#91A0;
   // UNICODE_TO_GBK[36059] := 16#E16C;
   // UNICODE_TO_GBK[36060] := 16#91A1;
   // UNICODE_TO_GBK[36061] := 16#E16D;
   // UNICODE_TO_GBK[36062] := 16#91A2;
   // UNICODE_TO_GBK[36063] := 16#F5B0;
   // UNICODE_TO_GBK[36064] := 16#91A3;
   // UNICODE_TO_GBK[36065] := 16#F5B1;
   // UNICODE_TO_GBK[36066] := 16#91A4;
   // UNICODE_TO_GBK[36067] := 16#E16E;
   // UNICODE_TO_GBK[36068] := 16#91A5;
   // UNICODE_TO_GBK[36069] := 16#E16F;
   // UNICODE_TO_GBK[36070] := 16#91A6;
   // UNICODE_TO_GBK[36071] := 16#E170;
   // UNICODE_TO_GBK[36072] := 16#91A7;
   // UNICODE_TO_GBK[36073] := 16#E171;
   // UNICODE_TO_GBK[36074] := 16#91A8;
   // UNICODE_TO_GBK[36075] := 16#E172;
   // UNICODE_TO_GBK[36076] := 16#91A9;
   // UNICODE_TO_GBK[36077] := 16#E173;
   // UNICODE_TO_GBK[36078] := 16#91AA;
   // UNICODE_TO_GBK[36079] := 16#F5B2;
   // UNICODE_TO_GBK[36080] := 16#91AB;
   // UNICODE_TO_GBK[36081] := 16#E174;
   // UNICODE_TO_GBK[36082] := 16#91AC;
   // UNICODE_TO_GBK[36083] := 16#E175;
   // UNICODE_TO_GBK[36084] := 16#91AD;
   // UNICODE_TO_GBK[36085] := 16#F5B3;
   // UNICODE_TO_GBK[36086] := 16#91AE;
   // UNICODE_TO_GBK[36087] := 16#F5B4;
   // UNICODE_TO_GBK[36088] := 16#91AF;
   // UNICODE_TO_GBK[36089] := 16#F5B5;
   // UNICODE_TO_GBK[36090] := 16#91B0;
   // UNICODE_TO_GBK[36091] := 16#E176;
   // UNICODE_TO_GBK[36092] := 16#91B1;
   // UNICODE_TO_GBK[36093] := 16#E177;
   // UNICODE_TO_GBK[36094] := 16#91B2;
   // UNICODE_TO_GBK[36095] := 16#E178;
   // UNICODE_TO_GBK[36096] := 16#91B3;
   // UNICODE_TO_GBK[36097] := 16#E179;
   // UNICODE_TO_GBK[36098] := 16#91B4;
   // UNICODE_TO_GBK[36099] := 16#F5B7;
   // UNICODE_TO_GBK[36100] := 16#91B5;
   // UNICODE_TO_GBK[36101] := 16#F5B6;
   // UNICODE_TO_GBK[36102] := 16#91B6;
   // UNICODE_TO_GBK[36103] := 16#E17A;
   // UNICODE_TO_GBK[36104] := 16#91B7;
   // UNICODE_TO_GBK[36105] := 16#E17B;
   // UNICODE_TO_GBK[36106] := 16#91B8;
   // UNICODE_TO_GBK[36107] := 16#E17C;
   // UNICODE_TO_GBK[36108] := 16#91B9;
   // UNICODE_TO_GBK[36109] := 16#E17D;
   // UNICODE_TO_GBK[36110] := 16#91BA;
   // UNICODE_TO_GBK[36111] := 16#F5B8;
   // UNICODE_TO_GBK[36112] := 16#91BB;
   // UNICODE_TO_GBK[36113] := 16#E17E;
   // UNICODE_TO_GBK[36114] := 16#91BC;
   // UNICODE_TO_GBK[36115] := 16#E180;
   // UNICODE_TO_GBK[36116] := 16#91BD;
   // UNICODE_TO_GBK[36117] := 16#E181;
   // UNICODE_TO_GBK[36118] := 16#91BE;
   // UNICODE_TO_GBK[36119] := 16#E182;
   // UNICODE_TO_GBK[36120] := 16#91BF;
   // UNICODE_TO_GBK[36121] := 16#E183;
   // UNICODE_TO_GBK[36122] := 16#91C0;
   // UNICODE_TO_GBK[36123] := 16#E184;
   // UNICODE_TO_GBK[36124] := 16#91C1;
   // UNICODE_TO_GBK[36125] := 16#E185;
   // UNICODE_TO_GBK[36126] := 16#91C2;
   // UNICODE_TO_GBK[36127] := 16#E186;
   // UNICODE_TO_GBK[36128] := 16#91C3;
   // UNICODE_TO_GBK[36129] := 16#E187;
   // UNICODE_TO_GBK[36130] := 16#91C4;
   // UNICODE_TO_GBK[36131] := 16#E188;
   // UNICODE_TO_GBK[36132] := 16#91C5;
   // UNICODE_TO_GBK[36133] := 16#E189;
   // UNICODE_TO_GBK[36134] := 16#91C6;
   // UNICODE_TO_GBK[36135] := 16#E18A;
   // UNICODE_TO_GBK[36136] := 16#91C7;
   // UNICODE_TO_GBK[36137] := 16#B2C9;
   // UNICODE_TO_GBK[36138] := 16#91C8;
   // UNICODE_TO_GBK[36139] := 16#E18B;
   // UNICODE_TO_GBK[36140] := 16#91C9;
   // UNICODE_TO_GBK[36141] := 16#D3D4;
   // UNICODE_TO_GBK[36142] := 16#91CA;
   // UNICODE_TO_GBK[36143] := 16#CACD;
   // UNICODE_TO_GBK[36144] := 16#91CB;
   // UNICODE_TO_GBK[36145] := 16#E18C;
   // UNICODE_TO_GBK[36146] := 16#91CC;
   // UNICODE_TO_GBK[36147] := 16#C0EF;
   // UNICODE_TO_GBK[36148] := 16#91CD;
   // UNICODE_TO_GBK[36149] := 16#D6D8;
   // UNICODE_TO_GBK[36150] := 16#91CE;
   // UNICODE_TO_GBK[36151] := 16#D2B0;
   // UNICODE_TO_GBK[36152] := 16#91CF;
   // UNICODE_TO_GBK[36153] := 16#C1BF;
   // UNICODE_TO_GBK[36154] := 16#91D0;
   // UNICODE_TO_GBK[36155] := 16#E18D;
   // UNICODE_TO_GBK[36156] := 16#91D1;
   // UNICODE_TO_GBK[36157] := 16#BDF0;
   // UNICODE_TO_GBK[36158] := 16#91D2;
   // UNICODE_TO_GBK[36159] := 16#E18E;
   // UNICODE_TO_GBK[36160] := 16#91D3;
   // UNICODE_TO_GBK[36161] := 16#E18F;
   // UNICODE_TO_GBK[36162] := 16#91D4;
   // UNICODE_TO_GBK[36163] := 16#E190;
   // UNICODE_TO_GBK[36164] := 16#91D5;
   // UNICODE_TO_GBK[36165] := 16#E191;
   // UNICODE_TO_GBK[36166] := 16#91D6;
   // UNICODE_TO_GBK[36167] := 16#E192;
   // UNICODE_TO_GBK[36168] := 16#91D7;
   // UNICODE_TO_GBK[36169] := 16#E193;
   // UNICODE_TO_GBK[36170] := 16#91D8;
   // UNICODE_TO_GBK[36171] := 16#E194;
   // UNICODE_TO_GBK[36172] := 16#91D9;
   // UNICODE_TO_GBK[36173] := 16#E195;
   // UNICODE_TO_GBK[36174] := 16#91DA;
   // UNICODE_TO_GBK[36175] := 16#E196;
   // UNICODE_TO_GBK[36176] := 16#91DB;
   // UNICODE_TO_GBK[36177] := 16#E197;
   // UNICODE_TO_GBK[36178] := 16#91DC;
   // UNICODE_TO_GBK[36179] := 16#B8AA;
   // UNICODE_TO_GBK[36180] := 16#91DD;
   // UNICODE_TO_GBK[36181] := 16#E198;
   // UNICODE_TO_GBK[36182] := 16#91DE;
   // UNICODE_TO_GBK[36183] := 16#E199;
   // UNICODE_TO_GBK[36184] := 16#91DF;
   // UNICODE_TO_GBK[36185] := 16#E19A;
   // UNICODE_TO_GBK[36186] := 16#91E0;
   // UNICODE_TO_GBK[36187] := 16#E19B;
   // UNICODE_TO_GBK[36188] := 16#91E1;
   // UNICODE_TO_GBK[36189] := 16#E19C;
   // UNICODE_TO_GBK[36190] := 16#91E2;
   // UNICODE_TO_GBK[36191] := 16#E19D;
   // UNICODE_TO_GBK[36192] := 16#91E3;
   // UNICODE_TO_GBK[36193] := 16#E19E;
   // UNICODE_TO_GBK[36194] := 16#91E4;
   // UNICODE_TO_GBK[36195] := 16#E19F;
   // UNICODE_TO_GBK[36196] := 16#91E5;
   // UNICODE_TO_GBK[36197] := 16#E1A0;
   // UNICODE_TO_GBK[36198] := 16#91E6;
   // UNICODE_TO_GBK[36199] := 16#E240;
   // UNICODE_TO_GBK[36200] := 16#91E7;
   // UNICODE_TO_GBK[36201] := 16#E241;
   // UNICODE_TO_GBK[36202] := 16#91E8;
   // UNICODE_TO_GBK[36203] := 16#E242;
   // UNICODE_TO_GBK[36204] := 16#91E9;
   // UNICODE_TO_GBK[36205] := 16#E243;
   // UNICODE_TO_GBK[36206] := 16#91EA;
   // UNICODE_TO_GBK[36207] := 16#E244;
   // UNICODE_TO_GBK[36208] := 16#91EB;
   // UNICODE_TO_GBK[36209] := 16#E245;
   // UNICODE_TO_GBK[36210] := 16#91EC;
   // UNICODE_TO_GBK[36211] := 16#E246;
   // UNICODE_TO_GBK[36212] := 16#91ED;
   // UNICODE_TO_GBK[36213] := 16#E247;
   // UNICODE_TO_GBK[36214] := 16#91EE;
   // UNICODE_TO_GBK[36215] := 16#E248;
   // UNICODE_TO_GBK[36216] := 16#91EF;
   // UNICODE_TO_GBK[36217] := 16#E249;
   // UNICODE_TO_GBK[36218] := 16#91F0;
   // UNICODE_TO_GBK[36219] := 16#E24A;
   // UNICODE_TO_GBK[36220] := 16#91F1;
   // UNICODE_TO_GBK[36221] := 16#E24B;
   // UNICODE_TO_GBK[36222] := 16#91F2;
   // UNICODE_TO_GBK[36223] := 16#E24C;
   // UNICODE_TO_GBK[36224] := 16#91F3;
   // UNICODE_TO_GBK[36225] := 16#E24D;
   // UNICODE_TO_GBK[36226] := 16#91F4;
   // UNICODE_TO_GBK[36227] := 16#E24E;
   // UNICODE_TO_GBK[36228] := 16#91F5;
   // UNICODE_TO_GBK[36229] := 16#E24F;
   // UNICODE_TO_GBK[36230] := 16#91F6;
   // UNICODE_TO_GBK[36231] := 16#E250;
   // UNICODE_TO_GBK[36232] := 16#91F7;
   // UNICODE_TO_GBK[36233] := 16#E251;
   // UNICODE_TO_GBK[36234] := 16#91F8;
   // UNICODE_TO_GBK[36235] := 16#E252;
   // UNICODE_TO_GBK[36236] := 16#91F9;
   // UNICODE_TO_GBK[36237] := 16#E253;
   // UNICODE_TO_GBK[36238] := 16#91FA;
   // UNICODE_TO_GBK[36239] := 16#E254;
   // UNICODE_TO_GBK[36240] := 16#91FB;
   // UNICODE_TO_GBK[36241] := 16#E255;
   // UNICODE_TO_GBK[36242] := 16#91FC;
   // UNICODE_TO_GBK[36243] := 16#E256;
   // UNICODE_TO_GBK[36244] := 16#91FD;
   // UNICODE_TO_GBK[36245] := 16#E257;
   // UNICODE_TO_GBK[36246] := 16#91FE;
   // UNICODE_TO_GBK[36247] := 16#E258;
   // UNICODE_TO_GBK[36248] := 16#91FF;
   // UNICODE_TO_GBK[36249] := 16#E259;
   // UNICODE_TO_GBK[36250] := 16#9200;
   // UNICODE_TO_GBK[36251] := 16#E25A;
   // UNICODE_TO_GBK[36252] := 16#9201;
   // UNICODE_TO_GBK[36253] := 16#E25B;
   // UNICODE_TO_GBK[36254] := 16#9202;
   // UNICODE_TO_GBK[36255] := 16#E25C;
   // UNICODE_TO_GBK[36256] := 16#9203;
   // UNICODE_TO_GBK[36257] := 16#E25D;
   // UNICODE_TO_GBK[36258] := 16#9204;
   // UNICODE_TO_GBK[36259] := 16#E25E;
   // UNICODE_TO_GBK[36260] := 16#9205;
   // UNICODE_TO_GBK[36261] := 16#E25F;
   // UNICODE_TO_GBK[36262] := 16#9206;
   // UNICODE_TO_GBK[36263] := 16#E260;
   // UNICODE_TO_GBK[36264] := 16#9207;
   // UNICODE_TO_GBK[36265] := 16#E261;
   // UNICODE_TO_GBK[36266] := 16#9208;
   // UNICODE_TO_GBK[36267] := 16#E262;
   // UNICODE_TO_GBK[36268] := 16#9209;
   // UNICODE_TO_GBK[36269] := 16#E263;
   // UNICODE_TO_GBK[36270] := 16#920A;
   // UNICODE_TO_GBK[36271] := 16#E264;
   // UNICODE_TO_GBK[36272] := 16#920B;
   // UNICODE_TO_GBK[36273] := 16#E265;
   // UNICODE_TO_GBK[36274] := 16#920C;
   // UNICODE_TO_GBK[36275] := 16#E266;
   // UNICODE_TO_GBK[36276] := 16#920D;
   // UNICODE_TO_GBK[36277] := 16#E267;
   // UNICODE_TO_GBK[36278] := 16#920E;
   // UNICODE_TO_GBK[36279] := 16#E268;
   // UNICODE_TO_GBK[36280] := 16#920F;
   // UNICODE_TO_GBK[36281] := 16#E269;
   // UNICODE_TO_GBK[36282] := 16#9210;
   // UNICODE_TO_GBK[36283] := 16#E26A;
   // UNICODE_TO_GBK[36284] := 16#9211;
   // UNICODE_TO_GBK[36285] := 16#E26B;
   // UNICODE_TO_GBK[36286] := 16#9212;
   // UNICODE_TO_GBK[36287] := 16#E26C;
   // UNICODE_TO_GBK[36288] := 16#9213;
   // UNICODE_TO_GBK[36289] := 16#E26D;
   // UNICODE_TO_GBK[36290] := 16#9214;
   // UNICODE_TO_GBK[36291] := 16#E26E;
   // UNICODE_TO_GBK[36292] := 16#9215;
   // UNICODE_TO_GBK[36293] := 16#E26F;
   // UNICODE_TO_GBK[36294] := 16#9216;
   // UNICODE_TO_GBK[36295] := 16#E270;
   // UNICODE_TO_GBK[36296] := 16#9217;
   // UNICODE_TO_GBK[36297] := 16#E271;
   // UNICODE_TO_GBK[36298] := 16#9218;
   // UNICODE_TO_GBK[36299] := 16#E272;
   // UNICODE_TO_GBK[36300] := 16#9219;
   // UNICODE_TO_GBK[36301] := 16#E273;
   // UNICODE_TO_GBK[36302] := 16#921A;
   // UNICODE_TO_GBK[36303] := 16#E274;
   // UNICODE_TO_GBK[36304] := 16#921B;
   // UNICODE_TO_GBK[36305] := 16#E275;
   // UNICODE_TO_GBK[36306] := 16#921C;
   // UNICODE_TO_GBK[36307] := 16#E276;
   // UNICODE_TO_GBK[36308] := 16#921D;
   // UNICODE_TO_GBK[36309] := 16#E277;
   // UNICODE_TO_GBK[36310] := 16#921E;
   // UNICODE_TO_GBK[36311] := 16#E278;
   // UNICODE_TO_GBK[36312] := 16#921F;
   // UNICODE_TO_GBK[36313] := 16#E279;
   // UNICODE_TO_GBK[36314] := 16#9220;
   // UNICODE_TO_GBK[36315] := 16#E27A;
   // UNICODE_TO_GBK[36316] := 16#9221;
   // UNICODE_TO_GBK[36317] := 16#E27B;
   // UNICODE_TO_GBK[36318] := 16#9222;
   // UNICODE_TO_GBK[36319] := 16#E27C;
   // UNICODE_TO_GBK[36320] := 16#9223;
   // UNICODE_TO_GBK[36321] := 16#E27D;
   // UNICODE_TO_GBK[36322] := 16#9224;
   // UNICODE_TO_GBK[36323] := 16#E27E;
   // UNICODE_TO_GBK[36324] := 16#9225;
   // UNICODE_TO_GBK[36325] := 16#E280;
   // UNICODE_TO_GBK[36326] := 16#9226;
   // UNICODE_TO_GBK[36327] := 16#E281;
   // UNICODE_TO_GBK[36328] := 16#9227;
   // UNICODE_TO_GBK[36329] := 16#E282;
   // UNICODE_TO_GBK[36330] := 16#9228;
   // UNICODE_TO_GBK[36331] := 16#E283;
   // UNICODE_TO_GBK[36332] := 16#9229;
   // UNICODE_TO_GBK[36333] := 16#E284;
   // UNICODE_TO_GBK[36334] := 16#922A;
   // UNICODE_TO_GBK[36335] := 16#E285;
   // UNICODE_TO_GBK[36336] := 16#922B;
   // UNICODE_TO_GBK[36337] := 16#E286;
   // UNICODE_TO_GBK[36338] := 16#922C;
   // UNICODE_TO_GBK[36339] := 16#E287;
   // UNICODE_TO_GBK[36340] := 16#922D;
   // UNICODE_TO_GBK[36341] := 16#E288;
   // UNICODE_TO_GBK[36342] := 16#922E;
   // UNICODE_TO_GBK[36343] := 16#E289;
   // UNICODE_TO_GBK[36344] := 16#922F;
   // UNICODE_TO_GBK[36345] := 16#E28A;
   // UNICODE_TO_GBK[36346] := 16#9230;
   // UNICODE_TO_GBK[36347] := 16#E28B;
   // UNICODE_TO_GBK[36348] := 16#9231;
   // UNICODE_TO_GBK[36349] := 16#E28C;
   // UNICODE_TO_GBK[36350] := 16#9232;
   // UNICODE_TO_GBK[36351] := 16#E28D;
   // UNICODE_TO_GBK[36352] := 16#9233;
   // UNICODE_TO_GBK[36353] := 16#E28E;
   // UNICODE_TO_GBK[36354] := 16#9234;
   // UNICODE_TO_GBK[36355] := 16#E28F;
   // UNICODE_TO_GBK[36356] := 16#9235;
   // UNICODE_TO_GBK[36357] := 16#E290;
   // UNICODE_TO_GBK[36358] := 16#9236;
   // UNICODE_TO_GBK[36359] := 16#E291;
   // UNICODE_TO_GBK[36360] := 16#9237;
   // UNICODE_TO_GBK[36361] := 16#E292;
   // UNICODE_TO_GBK[36362] := 16#9238;
   // UNICODE_TO_GBK[36363] := 16#E293;
   // UNICODE_TO_GBK[36364] := 16#9239;
   // UNICODE_TO_GBK[36365] := 16#E294;
   // UNICODE_TO_GBK[36366] := 16#923A;
   // UNICODE_TO_GBK[36367] := 16#E295;
   // UNICODE_TO_GBK[36368] := 16#923B;
   // UNICODE_TO_GBK[36369] := 16#E296;
   // UNICODE_TO_GBK[36370] := 16#923C;
   // UNICODE_TO_GBK[36371] := 16#E297;
   // UNICODE_TO_GBK[36372] := 16#923D;
   // UNICODE_TO_GBK[36373] := 16#E298;
   // UNICODE_TO_GBK[36374] := 16#923E;
   // UNICODE_TO_GBK[36375] := 16#E299;
   // UNICODE_TO_GBK[36376] := 16#923F;
   // UNICODE_TO_GBK[36377] := 16#E29A;
   // UNICODE_TO_GBK[36378] := 16#9240;
   // UNICODE_TO_GBK[36379] := 16#E29B;
   // UNICODE_TO_GBK[36380] := 16#9241;
   // UNICODE_TO_GBK[36381] := 16#E29C;
   // UNICODE_TO_GBK[36382] := 16#9242;
   // UNICODE_TO_GBK[36383] := 16#E29D;
   // UNICODE_TO_GBK[36384] := 16#9243;
   // UNICODE_TO_GBK[36385] := 16#E29E;
   // UNICODE_TO_GBK[36386] := 16#9244;
   // UNICODE_TO_GBK[36387] := 16#E29F;
   // UNICODE_TO_GBK[36388] := 16#9245;
   // UNICODE_TO_GBK[36389] := 16#E2A0;
   // UNICODE_TO_GBK[36390] := 16#9246;
   // UNICODE_TO_GBK[36391] := 16#E340;
   // UNICODE_TO_GBK[36392] := 16#9247;
   // UNICODE_TO_GBK[36393] := 16#E341;
   // UNICODE_TO_GBK[36394] := 16#9248;
   // UNICODE_TO_GBK[36395] := 16#E342;
   // UNICODE_TO_GBK[36396] := 16#9249;
   // UNICODE_TO_GBK[36397] := 16#E343;
   // UNICODE_TO_GBK[36398] := 16#924A;
   // UNICODE_TO_GBK[36399] := 16#E344;
   // UNICODE_TO_GBK[36400] := 16#924B;
   // UNICODE_TO_GBK[36401] := 16#E345;
   // UNICODE_TO_GBK[36402] := 16#924C;
   // UNICODE_TO_GBK[36403] := 16#E346;
   // UNICODE_TO_GBK[36404] := 16#924D;
   // UNICODE_TO_GBK[36405] := 16#E347;
   // UNICODE_TO_GBK[36406] := 16#924E;
   // UNICODE_TO_GBK[36407] := 16#E348;
   // UNICODE_TO_GBK[36408] := 16#924F;
   // UNICODE_TO_GBK[36409] := 16#E349;
   // UNICODE_TO_GBK[36410] := 16#9250;
   // UNICODE_TO_GBK[36411] := 16#E34A;
   // UNICODE_TO_GBK[36412] := 16#9251;
   // UNICODE_TO_GBK[36413] := 16#E34B;
   // UNICODE_TO_GBK[36414] := 16#9252;
   // UNICODE_TO_GBK[36415] := 16#E34C;
   // UNICODE_TO_GBK[36416] := 16#9253;
   // UNICODE_TO_GBK[36417] := 16#E34D;
   // UNICODE_TO_GBK[36418] := 16#9254;
   // UNICODE_TO_GBK[36419] := 16#E34E;
   // UNICODE_TO_GBK[36420] := 16#9255;
   // UNICODE_TO_GBK[36421] := 16#E34F;
   // UNICODE_TO_GBK[36422] := 16#9256;
   // UNICODE_TO_GBK[36423] := 16#E350;
   // UNICODE_TO_GBK[36424] := 16#9257;
   // UNICODE_TO_GBK[36425] := 16#E351;
   // UNICODE_TO_GBK[36426] := 16#9258;
   // UNICODE_TO_GBK[36427] := 16#E352;
   // UNICODE_TO_GBK[36428] := 16#9259;
   // UNICODE_TO_GBK[36429] := 16#E353;
   // UNICODE_TO_GBK[36430] := 16#925A;
   // UNICODE_TO_GBK[36431] := 16#E354;
   // UNICODE_TO_GBK[36432] := 16#925B;
   // UNICODE_TO_GBK[36433] := 16#E355;
   // UNICODE_TO_GBK[36434] := 16#925C;
   // UNICODE_TO_GBK[36435] := 16#E356;
   // UNICODE_TO_GBK[36436] := 16#925D;
   // UNICODE_TO_GBK[36437] := 16#E357;
   // UNICODE_TO_GBK[36438] := 16#925E;
   // UNICODE_TO_GBK[36439] := 16#E358;
   // UNICODE_TO_GBK[36440] := 16#925F;
   // UNICODE_TO_GBK[36441] := 16#E359;
   // UNICODE_TO_GBK[36442] := 16#9260;
   // UNICODE_TO_GBK[36443] := 16#E35A;
   // UNICODE_TO_GBK[36444] := 16#9261;
   // UNICODE_TO_GBK[36445] := 16#E35B;
   // UNICODE_TO_GBK[36446] := 16#9262;
   // UNICODE_TO_GBK[36447] := 16#E35C;
   // UNICODE_TO_GBK[36448] := 16#9263;
   // UNICODE_TO_GBK[36449] := 16#E35D;
   // UNICODE_TO_GBK[36450] := 16#9264;
   // UNICODE_TO_GBK[36451] := 16#E35E;
   // UNICODE_TO_GBK[36452] := 16#9265;
   // UNICODE_TO_GBK[36453] := 16#E35F;
   // UNICODE_TO_GBK[36454] := 16#9266;
   // UNICODE_TO_GBK[36455] := 16#E360;
   // UNICODE_TO_GBK[36456] := 16#9267;
   // UNICODE_TO_GBK[36457] := 16#E361;
   // UNICODE_TO_GBK[36458] := 16#9268;
   // UNICODE_TO_GBK[36459] := 16#E362;
   // UNICODE_TO_GBK[36460] := 16#9269;
   // UNICODE_TO_GBK[36461] := 16#E363;
   // UNICODE_TO_GBK[36462] := 16#926A;
   // UNICODE_TO_GBK[36463] := 16#E364;
   // UNICODE_TO_GBK[36464] := 16#926B;
   // UNICODE_TO_GBK[36465] := 16#E365;
   // UNICODE_TO_GBK[36466] := 16#926C;
   // UNICODE_TO_GBK[36467] := 16#E366;
   // UNICODE_TO_GBK[36468] := 16#926D;
   // UNICODE_TO_GBK[36469] := 16#E367;
   // UNICODE_TO_GBK[36470] := 16#926E;
   // UNICODE_TO_GBK[36471] := 16#E368;
   // UNICODE_TO_GBK[36472] := 16#926F;
   // UNICODE_TO_GBK[36473] := 16#E369;
   // UNICODE_TO_GBK[36474] := 16#9270;
   // UNICODE_TO_GBK[36475] := 16#E36A;
   // UNICODE_TO_GBK[36476] := 16#9271;
   // UNICODE_TO_GBK[36477] := 16#E36B;
   // UNICODE_TO_GBK[36478] := 16#9272;
   // UNICODE_TO_GBK[36479] := 16#E36C;
   // UNICODE_TO_GBK[36480] := 16#9273;
   // UNICODE_TO_GBK[36481] := 16#E36D;
   // UNICODE_TO_GBK[36482] := 16#9274;
   // UNICODE_TO_GBK[36483] := 16#BCF8;
   // UNICODE_TO_GBK[36484] := 16#9275;
   // UNICODE_TO_GBK[36485] := 16#E36E;
   // UNICODE_TO_GBK[36486] := 16#9276;
   // UNICODE_TO_GBK[36487] := 16#E36F;
   // UNICODE_TO_GBK[36488] := 16#9277;
   // UNICODE_TO_GBK[36489] := 16#E370;
   // UNICODE_TO_GBK[36490] := 16#9278;
   // UNICODE_TO_GBK[36491] := 16#E371;
   // UNICODE_TO_GBK[36492] := 16#9279;
   // UNICODE_TO_GBK[36493] := 16#E372;
   // UNICODE_TO_GBK[36494] := 16#927A;
   // UNICODE_TO_GBK[36495] := 16#E373;
   // UNICODE_TO_GBK[36496] := 16#927B;
   // UNICODE_TO_GBK[36497] := 16#E374;
   // UNICODE_TO_GBK[36498] := 16#927C;
   // UNICODE_TO_GBK[36499] := 16#E375;
   // UNICODE_TO_GBK[36500] := 16#927D;
   // UNICODE_TO_GBK[36501] := 16#E376;
   // UNICODE_TO_GBK[36502] := 16#927E;
   // UNICODE_TO_GBK[36503] := 16#E377;
   // UNICODE_TO_GBK[36504] := 16#927F;
   // UNICODE_TO_GBK[36505] := 16#E378;
   // UNICODE_TO_GBK[36506] := 16#9280;
   // UNICODE_TO_GBK[36507] := 16#E379;
   // UNICODE_TO_GBK[36508] := 16#9281;
   // UNICODE_TO_GBK[36509] := 16#E37A;
   // UNICODE_TO_GBK[36510] := 16#9282;
   // UNICODE_TO_GBK[36511] := 16#E37B;
   // UNICODE_TO_GBK[36512] := 16#9283;
   // UNICODE_TO_GBK[36513] := 16#E37C;
   // UNICODE_TO_GBK[36514] := 16#9284;
   // UNICODE_TO_GBK[36515] := 16#E37D;
   // UNICODE_TO_GBK[36516] := 16#9285;
   // UNICODE_TO_GBK[36517] := 16#E37E;
   // UNICODE_TO_GBK[36518] := 16#9286;
   // UNICODE_TO_GBK[36519] := 16#E380;
   // UNICODE_TO_GBK[36520] := 16#9287;
   // UNICODE_TO_GBK[36521] := 16#E381;
   // UNICODE_TO_GBK[36522] := 16#9288;
   // UNICODE_TO_GBK[36523] := 16#E382;
   // UNICODE_TO_GBK[36524] := 16#9289;
   // UNICODE_TO_GBK[36525] := 16#E383;
   // UNICODE_TO_GBK[36526] := 16#928A;
   // UNICODE_TO_GBK[36527] := 16#E384;
   // UNICODE_TO_GBK[36528] := 16#928B;
   // UNICODE_TO_GBK[36529] := 16#E385;
   // UNICODE_TO_GBK[36530] := 16#928C;
   // UNICODE_TO_GBK[36531] := 16#E386;
   // UNICODE_TO_GBK[36532] := 16#928D;
   // UNICODE_TO_GBK[36533] := 16#E387;
   // UNICODE_TO_GBK[36534] := 16#928E;
   // UNICODE_TO_GBK[36535] := 16#F6C6;
   // UNICODE_TO_GBK[36536] := 16#928F;
   // UNICODE_TO_GBK[36537] := 16#E388;
   // UNICODE_TO_GBK[36538] := 16#9290;
   // UNICODE_TO_GBK[36539] := 16#E389;
   // UNICODE_TO_GBK[36540] := 16#9291;
   // UNICODE_TO_GBK[36541] := 16#E38A;
   // UNICODE_TO_GBK[36542] := 16#9292;
   // UNICODE_TO_GBK[36543] := 16#E38B;
   // UNICODE_TO_GBK[36544] := 16#9293;
   // UNICODE_TO_GBK[36545] := 16#E38C;
   // UNICODE_TO_GBK[36546] := 16#9294;
   // UNICODE_TO_GBK[36547] := 16#E38D;
   // UNICODE_TO_GBK[36548] := 16#9295;
   // UNICODE_TO_GBK[36549] := 16#E38E;
   // UNICODE_TO_GBK[36550] := 16#9296;
   // UNICODE_TO_GBK[36551] := 16#E38F;
   // UNICODE_TO_GBK[36552] := 16#9297;
   // UNICODE_TO_GBK[36553] := 16#E390;
   // UNICODE_TO_GBK[36554] := 16#9298;
   // UNICODE_TO_GBK[36555] := 16#E391;
   // UNICODE_TO_GBK[36556] := 16#9299;
   // UNICODE_TO_GBK[36557] := 16#E392;
   // UNICODE_TO_GBK[36558] := 16#929A;
   // UNICODE_TO_GBK[36559] := 16#E393;
   // UNICODE_TO_GBK[36560] := 16#929B;
   // UNICODE_TO_GBK[36561] := 16#E394;
   // UNICODE_TO_GBK[36562] := 16#929C;
   // UNICODE_TO_GBK[36563] := 16#E395;
   // UNICODE_TO_GBK[36564] := 16#929D;
   // UNICODE_TO_GBK[36565] := 16#E396;
   // UNICODE_TO_GBK[36566] := 16#929E;
   // UNICODE_TO_GBK[36567] := 16#E397;
   // UNICODE_TO_GBK[36568] := 16#929F;
   // UNICODE_TO_GBK[36569] := 16#E398;
   // UNICODE_TO_GBK[36570] := 16#92A0;
   // UNICODE_TO_GBK[36571] := 16#E399;
   // UNICODE_TO_GBK[36572] := 16#92A1;
   // UNICODE_TO_GBK[36573] := 16#E39A;
   // UNICODE_TO_GBK[36574] := 16#92A2;
   // UNICODE_TO_GBK[36575] := 16#E39B;
   // UNICODE_TO_GBK[36576] := 16#92A3;
   // UNICODE_TO_GBK[36577] := 16#E39C;
   // UNICODE_TO_GBK[36578] := 16#92A4;
   // UNICODE_TO_GBK[36579] := 16#E39D;
   // UNICODE_TO_GBK[36580] := 16#92A5;
   // UNICODE_TO_GBK[36581] := 16#E39E;
   // UNICODE_TO_GBK[36582] := 16#92A6;
   // UNICODE_TO_GBK[36583] := 16#E39F;
   // UNICODE_TO_GBK[36584] := 16#92A7;
   // UNICODE_TO_GBK[36585] := 16#E3A0;
   // UNICODE_TO_GBK[36586] := 16#92A8;
   // UNICODE_TO_GBK[36587] := 16#E440;
   // UNICODE_TO_GBK[36588] := 16#92A9;
   // UNICODE_TO_GBK[36589] := 16#E441;
   // UNICODE_TO_GBK[36590] := 16#92AA;
   // UNICODE_TO_GBK[36591] := 16#E442;
   // UNICODE_TO_GBK[36592] := 16#92AB;
   // UNICODE_TO_GBK[36593] := 16#E443;
   // UNICODE_TO_GBK[36594] := 16#92AC;
   // UNICODE_TO_GBK[36595] := 16#E444;
   // UNICODE_TO_GBK[36596] := 16#92AD;
   // UNICODE_TO_GBK[36597] := 16#E445;
   // UNICODE_TO_GBK[36598] := 16#92AE;
   // UNICODE_TO_GBK[36599] := 16#F6C7;
   // UNICODE_TO_GBK[36600] := 16#92AF;
   // UNICODE_TO_GBK[36601] := 16#E446;
   // UNICODE_TO_GBK[36602] := 16#92B0;
   // UNICODE_TO_GBK[36603] := 16#E447;
   // UNICODE_TO_GBK[36604] := 16#92B1;
   // UNICODE_TO_GBK[36605] := 16#E448;
   // UNICODE_TO_GBK[36606] := 16#92B2;
   // UNICODE_TO_GBK[36607] := 16#E449;
   // UNICODE_TO_GBK[36608] := 16#92B3;
   // UNICODE_TO_GBK[36609] := 16#E44A;
   // UNICODE_TO_GBK[36610] := 16#92B4;
   // UNICODE_TO_GBK[36611] := 16#E44B;
   // UNICODE_TO_GBK[36612] := 16#92B5;
   // UNICODE_TO_GBK[36613] := 16#E44C;
   // UNICODE_TO_GBK[36614] := 16#92B6;
   // UNICODE_TO_GBK[36615] := 16#E44D;
   // UNICODE_TO_GBK[36616] := 16#92B7;
   // UNICODE_TO_GBK[36617] := 16#E44E;
   // UNICODE_TO_GBK[36618] := 16#92B8;
   // UNICODE_TO_GBK[36619] := 16#E44F;
   // UNICODE_TO_GBK[36620] := 16#92B9;
   // UNICODE_TO_GBK[36621] := 16#E450;
   // UNICODE_TO_GBK[36622] := 16#92BA;
   // UNICODE_TO_GBK[36623] := 16#E451;
   // UNICODE_TO_GBK[36624] := 16#92BB;
   // UNICODE_TO_GBK[36625] := 16#E452;
   // UNICODE_TO_GBK[36626] := 16#92BC;
   // UNICODE_TO_GBK[36627] := 16#E453;
   // UNICODE_TO_GBK[36628] := 16#92BD;
   // UNICODE_TO_GBK[36629] := 16#E454;
   // UNICODE_TO_GBK[36630] := 16#92BE;
   // UNICODE_TO_GBK[36631] := 16#E455;
   // UNICODE_TO_GBK[36632] := 16#92BF;
   // UNICODE_TO_GBK[36633] := 16#E456;
   // UNICODE_TO_GBK[36634] := 16#92C0;
   // UNICODE_TO_GBK[36635] := 16#E457;
   // UNICODE_TO_GBK[36636] := 16#92C1;
   // UNICODE_TO_GBK[36637] := 16#E458;
   // UNICODE_TO_GBK[36638] := 16#92C2;
   // UNICODE_TO_GBK[36639] := 16#E459;
   // UNICODE_TO_GBK[36640] := 16#92C3;
   // UNICODE_TO_GBK[36641] := 16#E45A;
   // UNICODE_TO_GBK[36642] := 16#92C4;
   // UNICODE_TO_GBK[36643] := 16#E45B;
   // UNICODE_TO_GBK[36644] := 16#92C5;
   // UNICODE_TO_GBK[36645] := 16#E45C;
   // UNICODE_TO_GBK[36646] := 16#92C6;
   // UNICODE_TO_GBK[36647] := 16#E45D;
   // UNICODE_TO_GBK[36648] := 16#92C7;
   // UNICODE_TO_GBK[36649] := 16#E45E;
   // UNICODE_TO_GBK[36650] := 16#92C8;
   // UNICODE_TO_GBK[36651] := 16#F6C8;
   // UNICODE_TO_GBK[36652] := 16#92C9;
   // UNICODE_TO_GBK[36653] := 16#E45F;
   // UNICODE_TO_GBK[36654] := 16#92CA;
   // UNICODE_TO_GBK[36655] := 16#E460;
   // UNICODE_TO_GBK[36656] := 16#92CB;
   // UNICODE_TO_GBK[36657] := 16#E461;
   // UNICODE_TO_GBK[36658] := 16#92CC;
   // UNICODE_TO_GBK[36659] := 16#E462;
   // UNICODE_TO_GBK[36660] := 16#92CD;
   // UNICODE_TO_GBK[36661] := 16#E463;
   // UNICODE_TO_GBK[36662] := 16#92CE;
   // UNICODE_TO_GBK[36663] := 16#E464;
   // UNICODE_TO_GBK[36664] := 16#92CF;
   // UNICODE_TO_GBK[36665] := 16#E465;
   // UNICODE_TO_GBK[36666] := 16#92D0;
   // UNICODE_TO_GBK[36667] := 16#E466;
   // UNICODE_TO_GBK[36668] := 16#92D1;
   // UNICODE_TO_GBK[36669] := 16#E467;
   // UNICODE_TO_GBK[36670] := 16#92D2;
   // UNICODE_TO_GBK[36671] := 16#E468;
   // UNICODE_TO_GBK[36672] := 16#92D3;
   // UNICODE_TO_GBK[36673] := 16#E469;
   // UNICODE_TO_GBK[36674] := 16#92D4;
   // UNICODE_TO_GBK[36675] := 16#E46A;
   // UNICODE_TO_GBK[36676] := 16#92D5;
   // UNICODE_TO_GBK[36677] := 16#E46B;
   // UNICODE_TO_GBK[36678] := 16#92D6;
   // UNICODE_TO_GBK[36679] := 16#E46C;
   // UNICODE_TO_GBK[36680] := 16#92D7;
   // UNICODE_TO_GBK[36681] := 16#E46D;
   // UNICODE_TO_GBK[36682] := 16#92D8;
   // UNICODE_TO_GBK[36683] := 16#E46E;
   // UNICODE_TO_GBK[36684] := 16#92D9;
   // UNICODE_TO_GBK[36685] := 16#E46F;
   // UNICODE_TO_GBK[36686] := 16#92DA;
   // UNICODE_TO_GBK[36687] := 16#E470;
   // UNICODE_TO_GBK[36688] := 16#92DB;
   // UNICODE_TO_GBK[36689] := 16#E471;
   // UNICODE_TO_GBK[36690] := 16#92DC;
   // UNICODE_TO_GBK[36691] := 16#E472;
   // UNICODE_TO_GBK[36692] := 16#92DD;
   // UNICODE_TO_GBK[36693] := 16#E473;
   // UNICODE_TO_GBK[36694] := 16#92DE;
   // UNICODE_TO_GBK[36695] := 16#E474;
   // UNICODE_TO_GBK[36696] := 16#92DF;
   // UNICODE_TO_GBK[36697] := 16#E475;
   // UNICODE_TO_GBK[36698] := 16#92E0;
   // UNICODE_TO_GBK[36699] := 16#E476;
   // UNICODE_TO_GBK[36700] := 16#92E1;
   // UNICODE_TO_GBK[36701] := 16#E477;
   // UNICODE_TO_GBK[36702] := 16#92E2;
   // UNICODE_TO_GBK[36703] := 16#E478;
   // UNICODE_TO_GBK[36704] := 16#92E3;
   // UNICODE_TO_GBK[36705] := 16#E479;
   // UNICODE_TO_GBK[36706] := 16#92E4;
   // UNICODE_TO_GBK[36707] := 16#E47A;
   // UNICODE_TO_GBK[36708] := 16#92E5;
   // UNICODE_TO_GBK[36709] := 16#E47B;
   // UNICODE_TO_GBK[36710] := 16#92E6;
   // UNICODE_TO_GBK[36711] := 16#E47C;
   // UNICODE_TO_GBK[36712] := 16#92E7;
   // UNICODE_TO_GBK[36713] := 16#E47D;
   // UNICODE_TO_GBK[36714] := 16#92E8;
   // UNICODE_TO_GBK[36715] := 16#E47E;
   // UNICODE_TO_GBK[36716] := 16#92E9;
   // UNICODE_TO_GBK[36717] := 16#E480;
   // UNICODE_TO_GBK[36718] := 16#92EA;
   // UNICODE_TO_GBK[36719] := 16#E481;
   // UNICODE_TO_GBK[36720] := 16#92EB;
   // UNICODE_TO_GBK[36721] := 16#E482;
   // UNICODE_TO_GBK[36722] := 16#92EC;
   // UNICODE_TO_GBK[36723] := 16#E483;
   // UNICODE_TO_GBK[36724] := 16#92ED;
   // UNICODE_TO_GBK[36725] := 16#E484;
   // UNICODE_TO_GBK[36726] := 16#92EE;
   // UNICODE_TO_GBK[36727] := 16#E485;
   // UNICODE_TO_GBK[36728] := 16#92EF;
   // UNICODE_TO_GBK[36729] := 16#E486;
   // UNICODE_TO_GBK[36730] := 16#92F0;
   // UNICODE_TO_GBK[36731] := 16#E487;
   // UNICODE_TO_GBK[36732] := 16#92F1;
   // UNICODE_TO_GBK[36733] := 16#E488;
   // UNICODE_TO_GBK[36734] := 16#92F2;
   // UNICODE_TO_GBK[36735] := 16#E489;
   // UNICODE_TO_GBK[36736] := 16#92F3;
   // UNICODE_TO_GBK[36737] := 16#E48A;
   // UNICODE_TO_GBK[36738] := 16#92F4;
   // UNICODE_TO_GBK[36739] := 16#E48B;
   // UNICODE_TO_GBK[36740] := 16#92F5;
   // UNICODE_TO_GBK[36741] := 16#E48C;
   // UNICODE_TO_GBK[36742] := 16#92F6;
   // UNICODE_TO_GBK[36743] := 16#E48D;
   // UNICODE_TO_GBK[36744] := 16#92F7;
   // UNICODE_TO_GBK[36745] := 16#E48E;
   // UNICODE_TO_GBK[36746] := 16#92F8;
   // UNICODE_TO_GBK[36747] := 16#E48F;
   // UNICODE_TO_GBK[36748] := 16#92F9;
   // UNICODE_TO_GBK[36749] := 16#E490;
   // UNICODE_TO_GBK[36750] := 16#92FA;
   // UNICODE_TO_GBK[36751] := 16#E491;
   // UNICODE_TO_GBK[36752] := 16#92FB;
   // UNICODE_TO_GBK[36753] := 16#E492;
   // UNICODE_TO_GBK[36754] := 16#92FC;
   // UNICODE_TO_GBK[36755] := 16#E493;
   // UNICODE_TO_GBK[36756] := 16#92FD;
   // UNICODE_TO_GBK[36757] := 16#E494;
   // UNICODE_TO_GBK[36758] := 16#92FE;
   // UNICODE_TO_GBK[36759] := 16#E495;
   // UNICODE_TO_GBK[36760] := 16#92FF;
   // UNICODE_TO_GBK[36761] := 16#E496;
   // UNICODE_TO_GBK[36762] := 16#9300;
   // UNICODE_TO_GBK[36763] := 16#E497;
   // UNICODE_TO_GBK[36764] := 16#9301;
   // UNICODE_TO_GBK[36765] := 16#E498;
   // UNICODE_TO_GBK[36766] := 16#9302;
   // UNICODE_TO_GBK[36767] := 16#E499;
   // UNICODE_TO_GBK[36768] := 16#9303;
   // UNICODE_TO_GBK[36769] := 16#E49A;
   // UNICODE_TO_GBK[36770] := 16#9304;
   // UNICODE_TO_GBK[36771] := 16#E49B;
   // UNICODE_TO_GBK[36772] := 16#9305;
   // UNICODE_TO_GBK[36773] := 16#E49C;
   // UNICODE_TO_GBK[36774] := 16#9306;
   // UNICODE_TO_GBK[36775] := 16#E49D;
   // UNICODE_TO_GBK[36776] := 16#9307;
   // UNICODE_TO_GBK[36777] := 16#E49E;
   // UNICODE_TO_GBK[36778] := 16#9308;
   // UNICODE_TO_GBK[36779] := 16#E49F;
   // UNICODE_TO_GBK[36780] := 16#9309;
   // UNICODE_TO_GBK[36781] := 16#E4A0;
   // UNICODE_TO_GBK[36782] := 16#930A;
   // UNICODE_TO_GBK[36783] := 16#E540;
   // UNICODE_TO_GBK[36784] := 16#930B;
   // UNICODE_TO_GBK[36785] := 16#E541;
   // UNICODE_TO_GBK[36786] := 16#930C;
   // UNICODE_TO_GBK[36787] := 16#E542;
   // UNICODE_TO_GBK[36788] := 16#930D;
   // UNICODE_TO_GBK[36789] := 16#E543;
   // UNICODE_TO_GBK[36790] := 16#930E;
   // UNICODE_TO_GBK[36791] := 16#E544;
   // UNICODE_TO_GBK[36792] := 16#930F;
   // UNICODE_TO_GBK[36793] := 16#E545;
   // UNICODE_TO_GBK[36794] := 16#9310;
   // UNICODE_TO_GBK[36795] := 16#E546;
   // UNICODE_TO_GBK[36796] := 16#9311;
   // UNICODE_TO_GBK[36797] := 16#E547;
   // UNICODE_TO_GBK[36798] := 16#9312;
   // UNICODE_TO_GBK[36799] := 16#E548;
   // UNICODE_TO_GBK[36800] := 16#9313;
   // UNICODE_TO_GBK[36801] := 16#E549;
   // UNICODE_TO_GBK[36802] := 16#9314;
   // UNICODE_TO_GBK[36803] := 16#E54A;
   // UNICODE_TO_GBK[36804] := 16#9315;
   // UNICODE_TO_GBK[36805] := 16#E54B;
   // UNICODE_TO_GBK[36806] := 16#9316;
   // UNICODE_TO_GBK[36807] := 16#E54C;
   // UNICODE_TO_GBK[36808] := 16#9317;
   // UNICODE_TO_GBK[36809] := 16#E54D;
   // UNICODE_TO_GBK[36810] := 16#9318;
   // UNICODE_TO_GBK[36811] := 16#E54E;
   // UNICODE_TO_GBK[36812] := 16#9319;
   // UNICODE_TO_GBK[36813] := 16#E54F;
   // UNICODE_TO_GBK[36814] := 16#931A;
   // UNICODE_TO_GBK[36815] := 16#E550;
   // UNICODE_TO_GBK[36816] := 16#931B;
   // UNICODE_TO_GBK[36817] := 16#E551;
   // UNICODE_TO_GBK[36818] := 16#931C;
   // UNICODE_TO_GBK[36819] := 16#E552;
   // UNICODE_TO_GBK[36820] := 16#931D;
   // UNICODE_TO_GBK[36821] := 16#E553;
   // UNICODE_TO_GBK[36822] := 16#931E;
   // UNICODE_TO_GBK[36823] := 16#E554;
   // UNICODE_TO_GBK[36824] := 16#931F;
   // UNICODE_TO_GBK[36825] := 16#E555;
   // UNICODE_TO_GBK[36826] := 16#9320;
   // UNICODE_TO_GBK[36827] := 16#E556;
   // UNICODE_TO_GBK[36828] := 16#9321;
   // UNICODE_TO_GBK[36829] := 16#E557;
   // UNICODE_TO_GBK[36830] := 16#9322;
   // UNICODE_TO_GBK[36831] := 16#E558;
   // UNICODE_TO_GBK[36832] := 16#9323;
   // UNICODE_TO_GBK[36833] := 16#E559;
   // UNICODE_TO_GBK[36834] := 16#9324;
   // UNICODE_TO_GBK[36835] := 16#E55A;
   // UNICODE_TO_GBK[36836] := 16#9325;
   // UNICODE_TO_GBK[36837] := 16#E55B;
   // UNICODE_TO_GBK[36838] := 16#9326;
   // UNICODE_TO_GBK[36839] := 16#E55C;
   // UNICODE_TO_GBK[36840] := 16#9327;
   // UNICODE_TO_GBK[36841] := 16#E55D;
   // UNICODE_TO_GBK[36842] := 16#9328;
   // UNICODE_TO_GBK[36843] := 16#E55E;
   // UNICODE_TO_GBK[36844] := 16#9329;
   // UNICODE_TO_GBK[36845] := 16#E55F;
   // UNICODE_TO_GBK[36846] := 16#932A;
   // UNICODE_TO_GBK[36847] := 16#E560;
   // UNICODE_TO_GBK[36848] := 16#932B;
   // UNICODE_TO_GBK[36849] := 16#E561;
   // UNICODE_TO_GBK[36850] := 16#932C;
   // UNICODE_TO_GBK[36851] := 16#E562;
   // UNICODE_TO_GBK[36852] := 16#932D;
   // UNICODE_TO_GBK[36853] := 16#E563;
   // UNICODE_TO_GBK[36854] := 16#932E;
   // UNICODE_TO_GBK[36855] := 16#E564;
   // UNICODE_TO_GBK[36856] := 16#932F;
   // UNICODE_TO_GBK[36857] := 16#E565;
   // UNICODE_TO_GBK[36858] := 16#9330;
   // UNICODE_TO_GBK[36859] := 16#E566;
   // UNICODE_TO_GBK[36860] := 16#9331;
   // UNICODE_TO_GBK[36861] := 16#E567;
   // UNICODE_TO_GBK[36862] := 16#9332;
   // UNICODE_TO_GBK[36863] := 16#E568;
   // UNICODE_TO_GBK[36864] := 16#9333;
   // UNICODE_TO_GBK[36865] := 16#E569;
   // UNICODE_TO_GBK[36866] := 16#9334;
   // UNICODE_TO_GBK[36867] := 16#E56A;
   // UNICODE_TO_GBK[36868] := 16#9335;
   // UNICODE_TO_GBK[36869] := 16#E56B;
   // UNICODE_TO_GBK[36870] := 16#9336;
   // UNICODE_TO_GBK[36871] := 16#E56C;
   // UNICODE_TO_GBK[36872] := 16#9337;
   // UNICODE_TO_GBK[36873] := 16#E56D;
   // UNICODE_TO_GBK[36874] := 16#9338;
   // UNICODE_TO_GBK[36875] := 16#E56E;
   // UNICODE_TO_GBK[36876] := 16#9339;
   // UNICODE_TO_GBK[36877] := 16#E56F;
   // UNICODE_TO_GBK[36878] := 16#933A;
   // UNICODE_TO_GBK[36879] := 16#E570;
   // UNICODE_TO_GBK[36880] := 16#933B;
   // UNICODE_TO_GBK[36881] := 16#E571;
   // UNICODE_TO_GBK[36882] := 16#933C;
   // UNICODE_TO_GBK[36883] := 16#E572;
   // UNICODE_TO_GBK[36884] := 16#933D;
   // UNICODE_TO_GBK[36885] := 16#E573;
   // UNICODE_TO_GBK[36886] := 16#933E;
   // UNICODE_TO_GBK[36887] := 16#F6C9;
   // UNICODE_TO_GBK[36888] := 16#933F;
   // UNICODE_TO_GBK[36889] := 16#E574;
   // UNICODE_TO_GBK[36890] := 16#9340;
   // UNICODE_TO_GBK[36891] := 16#E575;
   // UNICODE_TO_GBK[36892] := 16#9341;
   // UNICODE_TO_GBK[36893] := 16#E576;
   // UNICODE_TO_GBK[36894] := 16#9342;
   // UNICODE_TO_GBK[36895] := 16#E577;
   // UNICODE_TO_GBK[36896] := 16#9343;
   // UNICODE_TO_GBK[36897] := 16#E578;
   // UNICODE_TO_GBK[36898] := 16#9344;
   // UNICODE_TO_GBK[36899] := 16#E579;
   // UNICODE_TO_GBK[36900] := 16#9345;
   // UNICODE_TO_GBK[36901] := 16#E57A;
   // UNICODE_TO_GBK[36902] := 16#9346;
   // UNICODE_TO_GBK[36903] := 16#E57B;
   // UNICODE_TO_GBK[36904] := 16#9347;
   // UNICODE_TO_GBK[36905] := 16#E57C;
   // UNICODE_TO_GBK[36906] := 16#9348;
   // UNICODE_TO_GBK[36907] := 16#E57D;
   // UNICODE_TO_GBK[36908] := 16#9349;
   // UNICODE_TO_GBK[36909] := 16#E57E;
   // UNICODE_TO_GBK[36910] := 16#934A;
   // UNICODE_TO_GBK[36911] := 16#E580;
   // UNICODE_TO_GBK[36912] := 16#934B;
   // UNICODE_TO_GBK[36913] := 16#E581;
   // UNICODE_TO_GBK[36914] := 16#934C;
   // UNICODE_TO_GBK[36915] := 16#E582;
   // UNICODE_TO_GBK[36916] := 16#934D;
   // UNICODE_TO_GBK[36917] := 16#E583;
   // UNICODE_TO_GBK[36918] := 16#934E;
   // UNICODE_TO_GBK[36919] := 16#E584;
   // UNICODE_TO_GBK[36920] := 16#934F;
   // UNICODE_TO_GBK[36921] := 16#E585;
   // UNICODE_TO_GBK[36922] := 16#9350;
   // UNICODE_TO_GBK[36923] := 16#E586;
   // UNICODE_TO_GBK[36924] := 16#9351;
   // UNICODE_TO_GBK[36925] := 16#E587;
   // UNICODE_TO_GBK[36926] := 16#9352;
   // UNICODE_TO_GBK[36927] := 16#E588;
   // UNICODE_TO_GBK[36928] := 16#9353;
   // UNICODE_TO_GBK[36929] := 16#E589;
   // UNICODE_TO_GBK[36930] := 16#9354;
   // UNICODE_TO_GBK[36931] := 16#E58A;
   // UNICODE_TO_GBK[36932] := 16#9355;
   // UNICODE_TO_GBK[36933] := 16#E58B;
   // UNICODE_TO_GBK[36934] := 16#9356;
   // UNICODE_TO_GBK[36935] := 16#E58C;
   // UNICODE_TO_GBK[36936] := 16#9357;
   // UNICODE_TO_GBK[36937] := 16#E58D;
   // UNICODE_TO_GBK[36938] := 16#9358;
   // UNICODE_TO_GBK[36939] := 16#E58E;
   // UNICODE_TO_GBK[36940] := 16#9359;
   // UNICODE_TO_GBK[36941] := 16#E58F;
   // UNICODE_TO_GBK[36942] := 16#935A;
   // UNICODE_TO_GBK[36943] := 16#E590;
   // UNICODE_TO_GBK[36944] := 16#935B;
   // UNICODE_TO_GBK[36945] := 16#E591;
   // UNICODE_TO_GBK[36946] := 16#935C;
   // UNICODE_TO_GBK[36947] := 16#E592;
   // UNICODE_TO_GBK[36948] := 16#935D;
   // UNICODE_TO_GBK[36949] := 16#E593;
   // UNICODE_TO_GBK[36950] := 16#935E;
   // UNICODE_TO_GBK[36951] := 16#E594;
   // UNICODE_TO_GBK[36952] := 16#935F;
   // UNICODE_TO_GBK[36953] := 16#E595;
   // UNICODE_TO_GBK[36954] := 16#9360;
   // UNICODE_TO_GBK[36955] := 16#E596;
   // UNICODE_TO_GBK[36956] := 16#9361;
   // UNICODE_TO_GBK[36957] := 16#E597;
   // UNICODE_TO_GBK[36958] := 16#9362;
   // UNICODE_TO_GBK[36959] := 16#E598;
   // UNICODE_TO_GBK[36960] := 16#9363;
   // UNICODE_TO_GBK[36961] := 16#E599;
   // UNICODE_TO_GBK[36962] := 16#9364;
   // UNICODE_TO_GBK[36963] := 16#E59A;
   // UNICODE_TO_GBK[36964] := 16#9365;
   // UNICODE_TO_GBK[36965] := 16#E59B;
   // UNICODE_TO_GBK[36966] := 16#9366;
   // UNICODE_TO_GBK[36967] := 16#E59C;
   // UNICODE_TO_GBK[36968] := 16#9367;
   // UNICODE_TO_GBK[36969] := 16#E59D;
   // UNICODE_TO_GBK[36970] := 16#9368;
   // UNICODE_TO_GBK[36971] := 16#E59E;
   // UNICODE_TO_GBK[36972] := 16#9369;
   // UNICODE_TO_GBK[36973] := 16#E59F;
   // UNICODE_TO_GBK[36974] := 16#936A;
   // UNICODE_TO_GBK[36975] := 16#F6CA;
   // UNICODE_TO_GBK[36976] := 16#936B;
   // UNICODE_TO_GBK[36977] := 16#E5A0;
   // UNICODE_TO_GBK[36978] := 16#936C;
   // UNICODE_TO_GBK[36979] := 16#E640;
   // UNICODE_TO_GBK[36980] := 16#936D;
   // UNICODE_TO_GBK[36981] := 16#E641;
   // UNICODE_TO_GBK[36982] := 16#936E;
   // UNICODE_TO_GBK[36983] := 16#E642;
   // UNICODE_TO_GBK[36984] := 16#936F;
   // UNICODE_TO_GBK[36985] := 16#E643;
   // UNICODE_TO_GBK[36986] := 16#9370;
   // UNICODE_TO_GBK[36987] := 16#E644;
   // UNICODE_TO_GBK[36988] := 16#9371;
   // UNICODE_TO_GBK[36989] := 16#E645;
   // UNICODE_TO_GBK[36990] := 16#9372;
   // UNICODE_TO_GBK[36991] := 16#E646;
   // UNICODE_TO_GBK[36992] := 16#9373;
   // UNICODE_TO_GBK[36993] := 16#E647;
   // UNICODE_TO_GBK[36994] := 16#9374;
   // UNICODE_TO_GBK[36995] := 16#E648;
   // UNICODE_TO_GBK[36996] := 16#9375;
   // UNICODE_TO_GBK[36997] := 16#E649;
   // UNICODE_TO_GBK[36998] := 16#9376;
   // UNICODE_TO_GBK[36999] := 16#E64A;
   // UNICODE_TO_GBK[37000] := 16#9377;
   // UNICODE_TO_GBK[37001] := 16#E64B;
   // UNICODE_TO_GBK[37002] := 16#9378;
   // UNICODE_TO_GBK[37003] := 16#E64C;
   // UNICODE_TO_GBK[37004] := 16#9379;
   // UNICODE_TO_GBK[37005] := 16#E64D;
   // UNICODE_TO_GBK[37006] := 16#937A;
   // UNICODE_TO_GBK[37007] := 16#E64E;
   // UNICODE_TO_GBK[37008] := 16#937B;
   // UNICODE_TO_GBK[37009] := 16#E64F;
   // UNICODE_TO_GBK[37010] := 16#937C;
   // UNICODE_TO_GBK[37011] := 16#E650;
   // UNICODE_TO_GBK[37012] := 16#937D;
   // UNICODE_TO_GBK[37013] := 16#E651;
   // UNICODE_TO_GBK[37014] := 16#937E;
   // UNICODE_TO_GBK[37015] := 16#E652;
   // UNICODE_TO_GBK[37016] := 16#937F;
   // UNICODE_TO_GBK[37017] := 16#E653;
   // UNICODE_TO_GBK[37018] := 16#9380;
   // UNICODE_TO_GBK[37019] := 16#E654;
   // UNICODE_TO_GBK[37020] := 16#9381;
   // UNICODE_TO_GBK[37021] := 16#E655;
   // UNICODE_TO_GBK[37022] := 16#9382;
   // UNICODE_TO_GBK[37023] := 16#E656;
   // UNICODE_TO_GBK[37024] := 16#9383;
   // UNICODE_TO_GBK[37025] := 16#E657;
   // UNICODE_TO_GBK[37026] := 16#9384;
   // UNICODE_TO_GBK[37027] := 16#E658;
   // UNICODE_TO_GBK[37028] := 16#9385;
   // UNICODE_TO_GBK[37029] := 16#E659;
   // UNICODE_TO_GBK[37030] := 16#9386;
   // UNICODE_TO_GBK[37031] := 16#E65A;
   // UNICODE_TO_GBK[37032] := 16#9387;
   // UNICODE_TO_GBK[37033] := 16#E65B;
   // UNICODE_TO_GBK[37034] := 16#9388;
   // UNICODE_TO_GBK[37035] := 16#E65C;
   // UNICODE_TO_GBK[37036] := 16#9389;
   // UNICODE_TO_GBK[37037] := 16#E65D;
   // UNICODE_TO_GBK[37038] := 16#938A;
   // UNICODE_TO_GBK[37039] := 16#E65E;
   // UNICODE_TO_GBK[37040] := 16#938B;
   // UNICODE_TO_GBK[37041] := 16#E65F;
   // UNICODE_TO_GBK[37042] := 16#938C;
   // UNICODE_TO_GBK[37043] := 16#E660;
   // UNICODE_TO_GBK[37044] := 16#938D;
   // UNICODE_TO_GBK[37045] := 16#E661;
   // UNICODE_TO_GBK[37046] := 16#938E;
   // UNICODE_TO_GBK[37047] := 16#E662;
   // UNICODE_TO_GBK[37048] := 16#938F;
   // UNICODE_TO_GBK[37049] := 16#F6CC;
   // UNICODE_TO_GBK[37050] := 16#9390;
   // UNICODE_TO_GBK[37051] := 16#E663;
   // UNICODE_TO_GBK[37052] := 16#9391;
   // UNICODE_TO_GBK[37053] := 16#E664;
   // UNICODE_TO_GBK[37054] := 16#9392;
   // UNICODE_TO_GBK[37055] := 16#E665;
   // UNICODE_TO_GBK[37056] := 16#9393;
   // UNICODE_TO_GBK[37057] := 16#E666;
   // UNICODE_TO_GBK[37058] := 16#9394;
   // UNICODE_TO_GBK[37059] := 16#E667;
   // UNICODE_TO_GBK[37060] := 16#9395;
   // UNICODE_TO_GBK[37061] := 16#E668;
   // UNICODE_TO_GBK[37062] := 16#9396;
   // UNICODE_TO_GBK[37063] := 16#E669;
   // UNICODE_TO_GBK[37064] := 16#9397;
   // UNICODE_TO_GBK[37065] := 16#E66A;
   // UNICODE_TO_GBK[37066] := 16#9398;
   // UNICODE_TO_GBK[37067] := 16#E66B;
   // UNICODE_TO_GBK[37068] := 16#9399;
   // UNICODE_TO_GBK[37069] := 16#E66C;
   // UNICODE_TO_GBK[37070] := 16#939A;
   // UNICODE_TO_GBK[37071] := 16#E66D;
   // UNICODE_TO_GBK[37072] := 16#939B;
   // UNICODE_TO_GBK[37073] := 16#E66E;
   // UNICODE_TO_GBK[37074] := 16#939C;
   // UNICODE_TO_GBK[37075] := 16#E66F;
   // UNICODE_TO_GBK[37076] := 16#939D;
   // UNICODE_TO_GBK[37077] := 16#E670;
   // UNICODE_TO_GBK[37078] := 16#939E;
   // UNICODE_TO_GBK[37079] := 16#E671;
   // UNICODE_TO_GBK[37080] := 16#939F;
   // UNICODE_TO_GBK[37081] := 16#E672;
   // UNICODE_TO_GBK[37082] := 16#93A0;
   // UNICODE_TO_GBK[37083] := 16#E673;
   // UNICODE_TO_GBK[37084] := 16#93A1;
   // UNICODE_TO_GBK[37085] := 16#E674;
   // UNICODE_TO_GBK[37086] := 16#93A2;
   // UNICODE_TO_GBK[37087] := 16#E675;
   // UNICODE_TO_GBK[37088] := 16#93A3;
   // UNICODE_TO_GBK[37089] := 16#E676;
   // UNICODE_TO_GBK[37090] := 16#93A4;
   // UNICODE_TO_GBK[37091] := 16#E677;
   // UNICODE_TO_GBK[37092] := 16#93A5;
   // UNICODE_TO_GBK[37093] := 16#E678;
   // UNICODE_TO_GBK[37094] := 16#93A6;
   // UNICODE_TO_GBK[37095] := 16#E679;
   // UNICODE_TO_GBK[37096] := 16#93A7;
   // UNICODE_TO_GBK[37097] := 16#E67A;
   // UNICODE_TO_GBK[37098] := 16#93A8;
   // UNICODE_TO_GBK[37099] := 16#E67B;
   // UNICODE_TO_GBK[37100] := 16#93A9;
   // UNICODE_TO_GBK[37101] := 16#E67C;
   // UNICODE_TO_GBK[37102] := 16#93AA;
   // UNICODE_TO_GBK[37103] := 16#E67D;
   // UNICODE_TO_GBK[37104] := 16#93AB;
   // UNICODE_TO_GBK[37105] := 16#E67E;
   // UNICODE_TO_GBK[37106] := 16#93AC;
   // UNICODE_TO_GBK[37107] := 16#E680;
   // UNICODE_TO_GBK[37108] := 16#93AD;
   // UNICODE_TO_GBK[37109] := 16#E681;
   // UNICODE_TO_GBK[37110] := 16#93AE;
   // UNICODE_TO_GBK[37111] := 16#E682;
   // UNICODE_TO_GBK[37112] := 16#93AF;
   // UNICODE_TO_GBK[37113] := 16#E683;
   // UNICODE_TO_GBK[37114] := 16#93B0;
   // UNICODE_TO_GBK[37115] := 16#E684;
   // UNICODE_TO_GBK[37116] := 16#93B1;
   // UNICODE_TO_GBK[37117] := 16#E685;
   // UNICODE_TO_GBK[37118] := 16#93B2;
   // UNICODE_TO_GBK[37119] := 16#E686;
   // UNICODE_TO_GBK[37120] := 16#93B3;
   // UNICODE_TO_GBK[37121] := 16#E687;
   // UNICODE_TO_GBK[37122] := 16#93B4;
   // UNICODE_TO_GBK[37123] := 16#E688;
   // UNICODE_TO_GBK[37124] := 16#93B5;
   // UNICODE_TO_GBK[37125] := 16#E689;
   // UNICODE_TO_GBK[37126] := 16#93B6;
   // UNICODE_TO_GBK[37127] := 16#E68A;
   // UNICODE_TO_GBK[37128] := 16#93B7;
   // UNICODE_TO_GBK[37129] := 16#E68B;
   // UNICODE_TO_GBK[37130] := 16#93B8;
   // UNICODE_TO_GBK[37131] := 16#E68C;
   // UNICODE_TO_GBK[37132] := 16#93B9;
   // UNICODE_TO_GBK[37133] := 16#E68D;
   // UNICODE_TO_GBK[37134] := 16#93BA;
   // UNICODE_TO_GBK[37135] := 16#E68E;
   // UNICODE_TO_GBK[37136] := 16#93BB;
   // UNICODE_TO_GBK[37137] := 16#E68F;
   // UNICODE_TO_GBK[37138] := 16#93BC;
   // UNICODE_TO_GBK[37139] := 16#E690;
   // UNICODE_TO_GBK[37140] := 16#93BD;
   // UNICODE_TO_GBK[37141] := 16#E691;
   // UNICODE_TO_GBK[37142] := 16#93BE;
   // UNICODE_TO_GBK[37143] := 16#E692;
   // UNICODE_TO_GBK[37144] := 16#93BF;
   // UNICODE_TO_GBK[37145] := 16#E693;
   // UNICODE_TO_GBK[37146] := 16#93C0;
   // UNICODE_TO_GBK[37147] := 16#E694;
   // UNICODE_TO_GBK[37148] := 16#93C1;
   // UNICODE_TO_GBK[37149] := 16#E695;
   // UNICODE_TO_GBK[37150] := 16#93C2;
   // UNICODE_TO_GBK[37151] := 16#E696;
   // UNICODE_TO_GBK[37152] := 16#93C3;
   // UNICODE_TO_GBK[37153] := 16#E697;
   // UNICODE_TO_GBK[37154] := 16#93C4;
   // UNICODE_TO_GBK[37155] := 16#E698;
   // UNICODE_TO_GBK[37156] := 16#93C5;
   // UNICODE_TO_GBK[37157] := 16#E699;
   // UNICODE_TO_GBK[37158] := 16#93C6;
   // UNICODE_TO_GBK[37159] := 16#E69A;
   // UNICODE_TO_GBK[37160] := 16#93C7;
   // UNICODE_TO_GBK[37161] := 16#E69B;
   // UNICODE_TO_GBK[37162] := 16#93C8;
   // UNICODE_TO_GBK[37163] := 16#E69C;
   // UNICODE_TO_GBK[37164] := 16#93C9;
   // UNICODE_TO_GBK[37165] := 16#E69D;
   // UNICODE_TO_GBK[37166] := 16#93CA;
   // UNICODE_TO_GBK[37167] := 16#F6CB;
   // UNICODE_TO_GBK[37168] := 16#93CB;
   // UNICODE_TO_GBK[37169] := 16#E69E;
   // UNICODE_TO_GBK[37170] := 16#93CC;
   // UNICODE_TO_GBK[37171] := 16#E69F;
   // UNICODE_TO_GBK[37172] := 16#93CD;
   // UNICODE_TO_GBK[37173] := 16#E6A0;
   // UNICODE_TO_GBK[37174] := 16#93CE;
   // UNICODE_TO_GBK[37175] := 16#E740;
   // UNICODE_TO_GBK[37176] := 16#93CF;
   // UNICODE_TO_GBK[37177] := 16#E741;
   // UNICODE_TO_GBK[37178] := 16#93D0;
   // UNICODE_TO_GBK[37179] := 16#E742;
   // UNICODE_TO_GBK[37180] := 16#93D1;
   // UNICODE_TO_GBK[37181] := 16#E743;
   // UNICODE_TO_GBK[37182] := 16#93D2;
   // UNICODE_TO_GBK[37183] := 16#E744;
   // UNICODE_TO_GBK[37184] := 16#93D3;
   // UNICODE_TO_GBK[37185] := 16#E745;
   // UNICODE_TO_GBK[37186] := 16#93D4;
   // UNICODE_TO_GBK[37187] := 16#E746;
   // UNICODE_TO_GBK[37188] := 16#93D5;
   // UNICODE_TO_GBK[37189] := 16#E747;
   // UNICODE_TO_GBK[37190] := 16#93D6;
   // UNICODE_TO_GBK[37191] := 16#F7E9;
   // UNICODE_TO_GBK[37192] := 16#93D7;
   // UNICODE_TO_GBK[37193] := 16#E748;
   // UNICODE_TO_GBK[37194] := 16#93D8;
   // UNICODE_TO_GBK[37195] := 16#E749;
   // UNICODE_TO_GBK[37196] := 16#93D9;
   // UNICODE_TO_GBK[37197] := 16#E74A;
   // UNICODE_TO_GBK[37198] := 16#93DA;
   // UNICODE_TO_GBK[37199] := 16#E74B;
   // UNICODE_TO_GBK[37200] := 16#93DB;
   // UNICODE_TO_GBK[37201] := 16#E74C;
   // UNICODE_TO_GBK[37202] := 16#93DC;
   // UNICODE_TO_GBK[37203] := 16#E74D;
   // UNICODE_TO_GBK[37204] := 16#93DD;
   // UNICODE_TO_GBK[37205] := 16#E74E;
   // UNICODE_TO_GBK[37206] := 16#93DE;
   // UNICODE_TO_GBK[37207] := 16#E74F;
   // UNICODE_TO_GBK[37208] := 16#93DF;
   // UNICODE_TO_GBK[37209] := 16#E750;
   // UNICODE_TO_GBK[37210] := 16#93E0;
   // UNICODE_TO_GBK[37211] := 16#E751;
   // UNICODE_TO_GBK[37212] := 16#93E1;
   // UNICODE_TO_GBK[37213] := 16#E752;
   // UNICODE_TO_GBK[37214] := 16#93E2;
   // UNICODE_TO_GBK[37215] := 16#E753;
   // UNICODE_TO_GBK[37216] := 16#93E3;
   // UNICODE_TO_GBK[37217] := 16#E754;
   // UNICODE_TO_GBK[37218] := 16#93E4;
   // UNICODE_TO_GBK[37219] := 16#E755;
   // UNICODE_TO_GBK[37220] := 16#93E5;
   // UNICODE_TO_GBK[37221] := 16#E756;
   // UNICODE_TO_GBK[37222] := 16#93E6;
   // UNICODE_TO_GBK[37223] := 16#E757;
   // UNICODE_TO_GBK[37224] := 16#93E7;
   // UNICODE_TO_GBK[37225] := 16#E758;
   // UNICODE_TO_GBK[37226] := 16#93E8;
   // UNICODE_TO_GBK[37227] := 16#E759;
   // UNICODE_TO_GBK[37228] := 16#93E9;
   // UNICODE_TO_GBK[37229] := 16#E75A;
   // UNICODE_TO_GBK[37230] := 16#93EA;
   // UNICODE_TO_GBK[37231] := 16#E75B;
   // UNICODE_TO_GBK[37232] := 16#93EB;
   // UNICODE_TO_GBK[37233] := 16#E75C;
   // UNICODE_TO_GBK[37234] := 16#93EC;
   // UNICODE_TO_GBK[37235] := 16#E75D;
   // UNICODE_TO_GBK[37236] := 16#93ED;
   // UNICODE_TO_GBK[37237] := 16#E75E;
   // UNICODE_TO_GBK[37238] := 16#93EE;
   // UNICODE_TO_GBK[37239] := 16#E75F;
   // UNICODE_TO_GBK[37240] := 16#93EF;
   // UNICODE_TO_GBK[37241] := 16#E760;
   // UNICODE_TO_GBK[37242] := 16#93F0;
   // UNICODE_TO_GBK[37243] := 16#E761;
   // UNICODE_TO_GBK[37244] := 16#93F1;
   // UNICODE_TO_GBK[37245] := 16#E762;
   // UNICODE_TO_GBK[37246] := 16#93F2;
   // UNICODE_TO_GBK[37247] := 16#E763;
   // UNICODE_TO_GBK[37248] := 16#93F3;
   // UNICODE_TO_GBK[37249] := 16#E764;
   // UNICODE_TO_GBK[37250] := 16#93F4;
   // UNICODE_TO_GBK[37251] := 16#E765;
   // UNICODE_TO_GBK[37252] := 16#93F5;
   // UNICODE_TO_GBK[37253] := 16#E766;
   // UNICODE_TO_GBK[37254] := 16#93F6;
   // UNICODE_TO_GBK[37255] := 16#E767;
   // UNICODE_TO_GBK[37256] := 16#93F7;
   // UNICODE_TO_GBK[37257] := 16#E768;
   // UNICODE_TO_GBK[37258] := 16#93F8;
   // UNICODE_TO_GBK[37259] := 16#E769;
   // UNICODE_TO_GBK[37260] := 16#93F9;
   // UNICODE_TO_GBK[37261] := 16#E76A;
   // UNICODE_TO_GBK[37262] := 16#93FA;
   // UNICODE_TO_GBK[37263] := 16#E76B;
   // UNICODE_TO_GBK[37264] := 16#93FB;
   // UNICODE_TO_GBK[37265] := 16#E76C;
   // UNICODE_TO_GBK[37266] := 16#93FC;
   // UNICODE_TO_GBK[37267] := 16#E76D;
   // UNICODE_TO_GBK[37268] := 16#93FD;
   // UNICODE_TO_GBK[37269] := 16#E76E;
   // UNICODE_TO_GBK[37270] := 16#93FE;
   // UNICODE_TO_GBK[37271] := 16#E76F;
   // UNICODE_TO_GBK[37272] := 16#93FF;
   // UNICODE_TO_GBK[37273] := 16#E770;
   // UNICODE_TO_GBK[37274] := 16#9400;
   // UNICODE_TO_GBK[37275] := 16#E771;
   // UNICODE_TO_GBK[37276] := 16#9401;
   // UNICODE_TO_GBK[37277] := 16#E772;
   // UNICODE_TO_GBK[37278] := 16#9402;
   // UNICODE_TO_GBK[37279] := 16#E773;
   // UNICODE_TO_GBK[37280] := 16#9403;
   // UNICODE_TO_GBK[37281] := 16#E774;
   // UNICODE_TO_GBK[37282] := 16#9404;
   // UNICODE_TO_GBK[37283] := 16#E775;
   // UNICODE_TO_GBK[37284] := 16#9405;
   // UNICODE_TO_GBK[37285] := 16#E776;
   // UNICODE_TO_GBK[37286] := 16#9406;
   // UNICODE_TO_GBK[37287] := 16#E777;
   // UNICODE_TO_GBK[37288] := 16#9407;
   // UNICODE_TO_GBK[37289] := 16#E778;
   // UNICODE_TO_GBK[37290] := 16#9408;
   // UNICODE_TO_GBK[37291] := 16#E779;
   // UNICODE_TO_GBK[37292] := 16#9409;
   // UNICODE_TO_GBK[37293] := 16#E77A;
   // UNICODE_TO_GBK[37294] := 16#940A;
   // UNICODE_TO_GBK[37295] := 16#E77B;
   // UNICODE_TO_GBK[37296] := 16#940B;
   // UNICODE_TO_GBK[37297] := 16#E77C;
   // UNICODE_TO_GBK[37298] := 16#940C;
   // UNICODE_TO_GBK[37299] := 16#E77D;
   // UNICODE_TO_GBK[37300] := 16#940D;
   // UNICODE_TO_GBK[37301] := 16#E77E;
   // UNICODE_TO_GBK[37302] := 16#940E;
   // UNICODE_TO_GBK[37303] := 16#E780;
   // UNICODE_TO_GBK[37304] := 16#940F;
   // UNICODE_TO_GBK[37305] := 16#E781;
   // UNICODE_TO_GBK[37306] := 16#9410;
   // UNICODE_TO_GBK[37307] := 16#E782;
   // UNICODE_TO_GBK[37308] := 16#9411;
   // UNICODE_TO_GBK[37309] := 16#E783;
   // UNICODE_TO_GBK[37310] := 16#9412;
   // UNICODE_TO_GBK[37311] := 16#E784;
   // UNICODE_TO_GBK[37312] := 16#9413;
   // UNICODE_TO_GBK[37313] := 16#E785;
   // UNICODE_TO_GBK[37314] := 16#9414;
   // UNICODE_TO_GBK[37315] := 16#E786;
   // UNICODE_TO_GBK[37316] := 16#9415;
   // UNICODE_TO_GBK[37317] := 16#E787;
   // UNICODE_TO_GBK[37318] := 16#9416;
   // UNICODE_TO_GBK[37319] := 16#E788;
   // UNICODE_TO_GBK[37320] := 16#9417;
   // UNICODE_TO_GBK[37321] := 16#E789;
   // UNICODE_TO_GBK[37322] := 16#9418;
   // UNICODE_TO_GBK[37323] := 16#E78A;
   // UNICODE_TO_GBK[37324] := 16#9419;
   // UNICODE_TO_GBK[37325] := 16#E78B;
